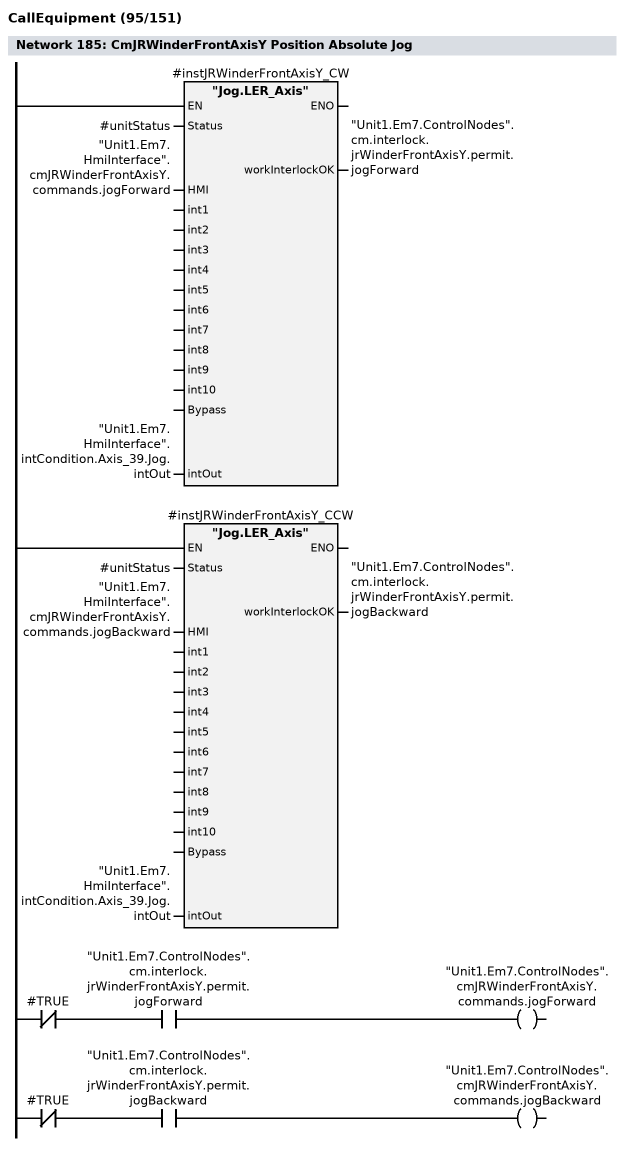
   RUNG wire#powerrail
      #instJRWinderFrontAxisY_CW(Status := #unitStatus, HMI := "Unit1.Em7.HmiInterface".cmJRWinderFrontAxisY.commands.jogForward, int1 :=, int2 :=, int3 :=, int4 :=, int5 :=, int6 :=, int7 :=, int8 :=, int9 :=, int10 :=, Bypass :=, intOut := "Unit1.Em7.HmiInterface".intCondition.Axis_39.Jog.intOut, workInterlockOK => "Unit1.Em7.ControlNodes".cm.interlock.jrWinderFrontAxisY.permit.jogForward)
   END_RUNG
   RUNG wire#powerrail
      #instJRWinderFrontAxisY_CCW(Status := #unitStatus, HMI := "Unit1.Em7.HmiInterface".cmJRWinderFrontAxisY.commands.jogBackward, int1 :=, int2 :=, int3 :=, int4 :=, int5 :=, int6 :=, int7 :=, int8 :=, int9 :=, int10 :=, Bypass :=, intOut := "Unit1.Em7.HmiInterface".intCondition.Axis_39.Jog.intOut, workInterlockOK => "Unit1.Em7.ControlNodes".cm.interlock.jrWinderFrontAxisY.permit.jogBackward)
   END_RUNG
   RUNG wire#powerrail
      I_Contact( #TRUE )
      Contact( "Unit1.Em7.ControlNodes".cm.interlock.jrWinderFrontAxisY.permit.jogForward )
      Coil( "Unit1.Em7.ControlNodes".cmJRWinderFrontAxisY.commands.jogForward )
   END_RUNG
   RUNG wire#powerrail
      I_Contact( #TRUE )
      Contact( "Unit1.Em7.ControlNodes".cm.interlock.jrWinderFrontAxisY.permit.jogBackward )
      Coil( "Unit1.Em7.ControlNodes".cmJRWinderFrontAxisY.commands.jogBackward )
   END_RUNG
   // the same network as SCL:
   #instJRWinderFrontAxisY_CW(Status := #unitStatus,   // "Jog.LER_Axis"
                           HMI := "Unit1.Em7.HmiInterface".cmJRWinderFrontAxisY.commands.jogForward,
                           intOut := "Unit1.Em7.HmiInterface".intCondition.Axis_39.Jog.intOut,
                           workInterlockOK => "Unit1.Em7.ControlNodes".cm.interlock.jrWinderFrontAxisY.permit.jogForward);
   #instJRWinderFrontAxisY_CCW(Status := #unitStatus,   // "Jog.LER_Axis"
                           HMI := "Unit1.Em7.HmiInterface".cmJRWinderFrontAxisY.commands.jogBackward,
                           intOut := "Unit1.Em7.HmiInterface".intCondition.Axis_39.Jog.intOut,
                           workInterlockOK => "Unit1.Em7.ControlNodes".cm.interlock.jrWinderFrontAxisY.permit.jogBackward);
   "Unit1.Em7.ControlNodes".cmJRWinderFrontAxisY.commands.jogForward := NOT #TRUE AND "Unit1.Em7.ControlNodes".cm.interlock.jrWinderFrontAxisY.permit.jogForward;
   "Unit1.Em7.ControlNodes".cmJRWinderFrontAxisY.commands.jogBackward := NOT #TRUE AND "Unit1.Em7.ControlNodes".cm.interlock.jrWinderFrontAxisY.permit.jogBackward;
END_REGION

REGION Network 186: CmJRWinderFrontAxisY Position Absolute Position0
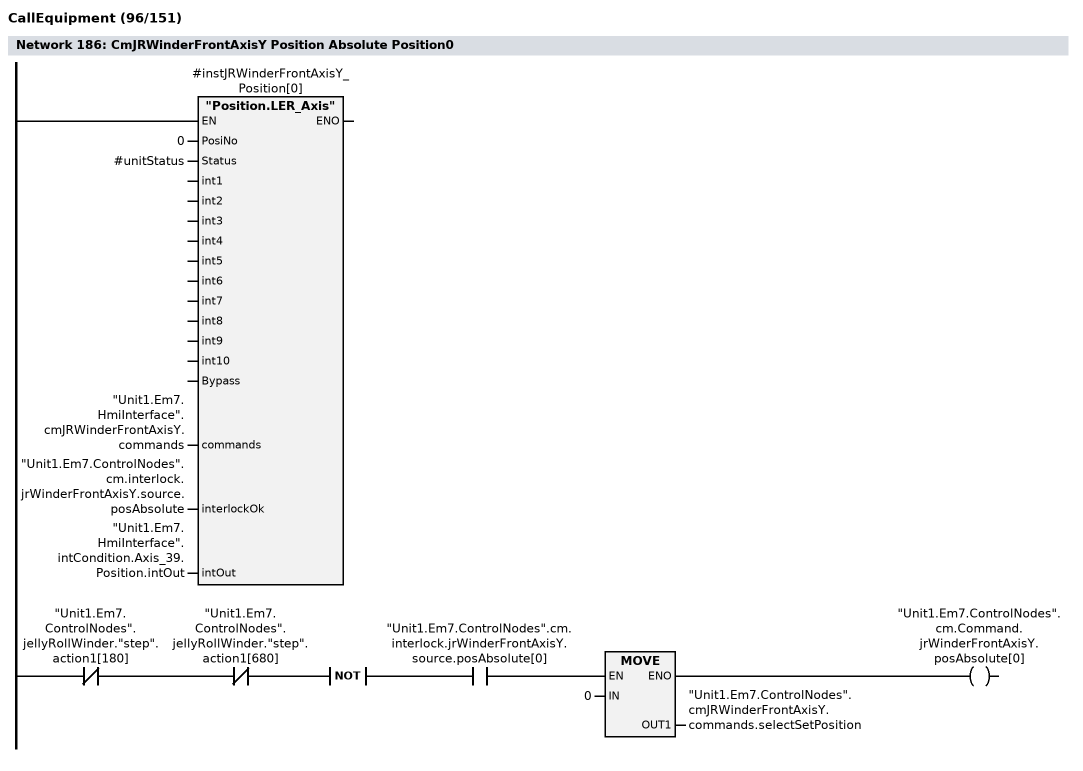
   RUNG wire#powerrail
      #instJRWinderFrontAxisY_Position[0](PosiNo := 0, Status := #unitStatus, int1 :=, int2 :=, int3 :=, int4 :=, int5 :=, int6 :=, int7 :=, int8 :=, int9 :=, int10 :=, Bypass :=, commands := "Unit1.Em7.HmiInterface".cmJRWinderFrontAxisY.commands, interlockOk := "Unit1.Em7.ControlNodes".cm.interlock.jrWinderFrontAxisY.source.posAbsolute, intOut := "Unit1.Em7.HmiInterface".intCondition.Axis_39.Position.intOut)
   END_RUNG
   RUNG wire#powerrail
      I_Contact( "Unit1.Em7.ControlNodes".jellyRollWinder."step".action1[180] )
      I_Contact( "Unit1.Em7.ControlNodes".jellyRollWinder."step".action1[680] )
      Not()
      Contact( "Unit1.Em7.ControlNodes".cm.interlock.jrWinderFrontAxisY.source.posAbsolute[0] )
      Move(in := 0, out1 => "Unit1.Em7.ControlNodes".cmJRWinderFrontAxisY.commands.selectSetPosition)
      Coil( "Unit1.Em7.ControlNodes".cm.Command.jrWinderFrontAxisY.posAbsolute[0] )
   END_RUNG
   // the same network as SCL:
   #instJRWinderFrontAxisY_Position[0](PosiNo := 0,   // "Position.LER_Axis"
                           Status := #unitStatus,
                           commands := "Unit1.Em7.HmiInterface".cmJRWinderFrontAxisY.commands,
                           interlockOk := "Unit1.Em7.ControlNodes".cm.interlock.jrWinderFrontAxisY.source.posAbsolute,
                           intOut := "Unit1.Em7.HmiInterface".intCondition.Axis_39.Position.intOut);
   #_w1 := NOT (NOT "Unit1.Em7.ControlNodes".jellyRollWinder."step".action1[180] AND NOT "Unit1.Em7.ControlNodes".jellyRollWinder."step".action1[680]) AND "Unit1.Em7.ControlNodes".cm.interlock.jrWinderFrontAxisY.source.posAbsolute[0];
   IF #_w1 THEN "Unit1.Em7.ControlNodes".cmJRWinderFrontAxisY.commands.selectSetPosition := 0; END_IF;
   "Unit1.Em7.ControlNodes".cm.Command.jrWinderFrontAxisY.posAbsolute[0] := #_w1;
END_REGION

REGION Network 187: CmJRWinderFrontAxisY Position Absolute Position1
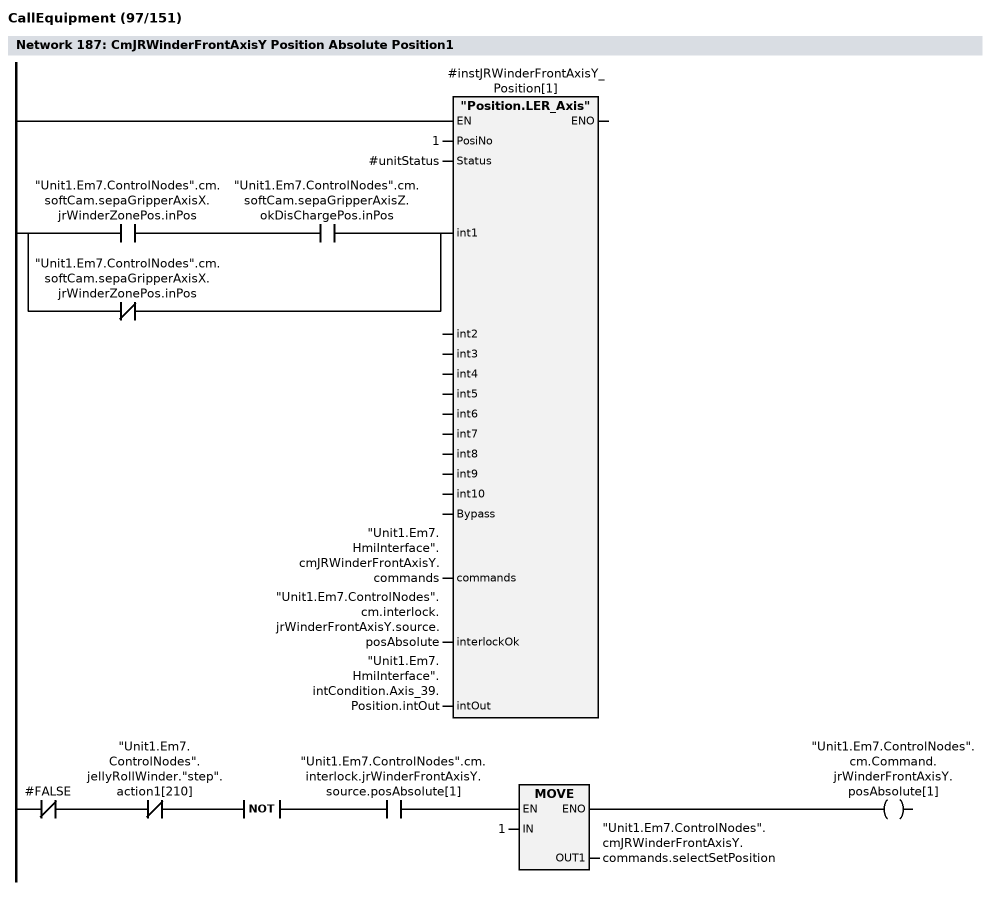
   RUNG wire#powerrail
      #instJRWinderFrontAxisY_Position[1](int1 := wire#w1, PosiNo := 1, Status := #unitStatus, int2 :=, int3 :=, int4 :=, int5 :=, int6 :=, int7 :=, int8 :=, int9 :=, int10 :=, Bypass :=, commands := "Unit1.Em7.HmiInterface".cmJRWinderFrontAxisY.commands, interlockOk := "Unit1.Em7.ControlNodes".cm.interlock.jrWinderFrontAxisY.source.posAbsolute, intOut := "Unit1.Em7.HmiInterface".intCondition.Axis_39.Position.intOut)
   END_RUNG
   RUNG wire#powerrail
      Contact( "Unit1.Em7.ControlNodes".cm.softCam.sepaGripperAxisX.jrWinderZonePos.inPos )
      Contact( "Unit1.Em7.ControlNodes".cm.softCam.sepaGripperAxisZ.okDisChargePos.inPos )
   END_RUNG wire#w1
   RUNG wire#powerrail
      I_Contact( "Unit1.Em7.ControlNodes".cm.softCam.sepaGripperAxisX.jrWinderZonePos.inPos )
   END_RUNG wire#w1
   RUNG wire#powerrail
      I_Contact( #FALSE )
      I_Contact( "Unit1.Em7.ControlNodes".jellyRollWinder."step".action1[210] )
      Not()
      Contact( "Unit1.Em7.ControlNodes".cm.interlock.jrWinderFrontAxisY.source.posAbsolute[1] )
      Move(in := 1, out1 => "Unit1.Em7.ControlNodes".cmJRWinderFrontAxisY.commands.selectSetPosition)
      Coil( "Unit1.Em7.ControlNodes".cm.Command.jrWinderFrontAxisY.posAbsolute[1] )
   END_RUNG
   // the same network as SCL:
   #instJRWinderFrontAxisY_Position[1](PosiNo := 1,   // "Position.LER_Axis"
                           Status := #unitStatus,
                           int1 := ("Unit1.Em7.ControlNodes".cm.softCam.sepaGripperAxisX.jrWinderZonePos.inPos AND "Unit1.Em7.ControlNodes".cm.softCam.sepaGripperAxisZ.okDisChargePos.inPos) OR NOT "Unit1.Em7.ControlNodes".cm.softCam.sepaGripperAxisX.jrWinderZonePos.inPos,
                           commands := "Unit1.Em7.HmiInterface".cmJRWinderFrontAxisY.commands,
                           interlockOk := "Unit1.Em7.ControlNodes".cm.interlock.jrWinderFrontAxisY.source.posAbsolute,
                           intOut := "Unit1.Em7.HmiInterface".intCondition.Axis_39.Position.intOut);
   #_w1 := NOT (NOT #FALSE AND NOT "Unit1.Em7.ControlNodes".jellyRollWinder."step".action1[210]) AND "Unit1.Em7.ControlNodes".cm.interlock.jrWinderFrontAxisY.source.posAbsolute[1];
   IF #_w1 THEN "Unit1.Em7.ControlNodes".cmJRWinderFrontAxisY.commands.selectSetPosition := 1; END_IF;
   "Unit1.Em7.ControlNodes".cm.Command.jrWinderFrontAxisY.posAbsolute[1] := #_w1;
END_REGION

REGION Network 188: CmJRWinderFrontAxisY Position Absolute Position2
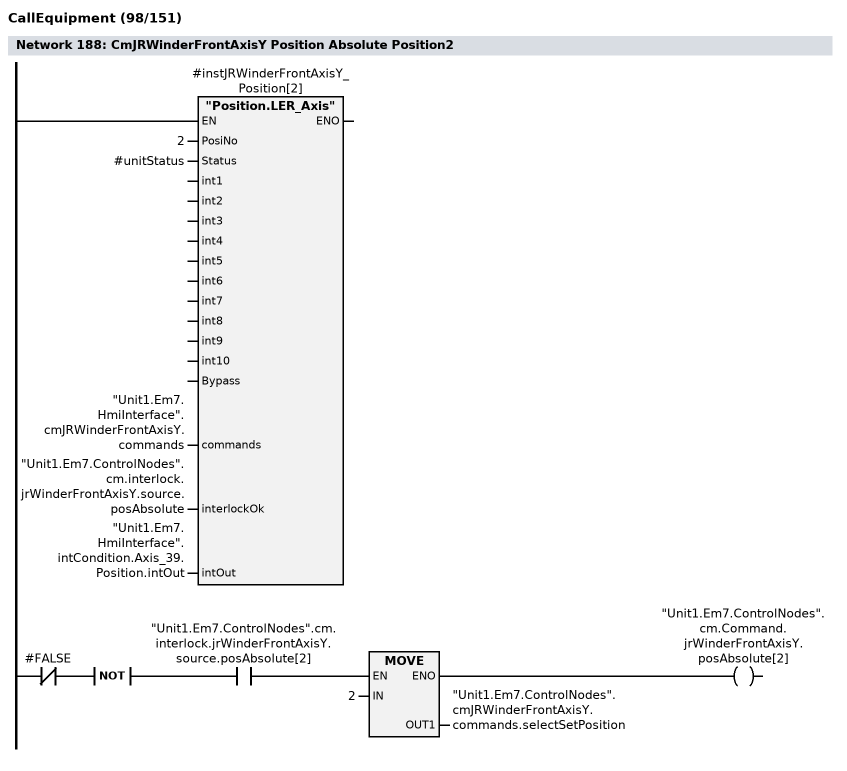
   RUNG wire#powerrail
      #instJRWinderFrontAxisY_Position[2](PosiNo := 2, Status := #unitStatus, int1 :=, int2 :=, int3 :=, int4 :=, int5 :=, int6 :=, int7 :=, int8 :=, int9 :=, int10 :=, Bypass :=, commands := "Unit1.Em7.HmiInterface".cmJRWinderFrontAxisY.commands, interlockOk := "Unit1.Em7.ControlNodes".cm.interlock.jrWinderFrontAxisY.source.posAbsolute, intOut := "Unit1.Em7.HmiInterface".intCondition.Axis_39.Position.intOut)
   END_RUNG
   RUNG wire#powerrail
      I_Contact( #FALSE )
      Not()
      Contact( "Unit1.Em7.ControlNodes".cm.interlock.jrWinderFrontAxisY.source.posAbsolute[2] )
      Move(in := 2, out1 => "Unit1.Em7.ControlNodes".cmJRWinderFrontAxisY.commands.selectSetPosition)
      Coil( "Unit1.Em7.ControlNodes".cm.Command.jrWinderFrontAxisY.posAbsolute[2] )
   END_RUNG
   // the same network as SCL:
   #instJRWinderFrontAxisY_Position[2](PosiNo := 2,   // "Position.LER_Axis"
                           Status := #unitStatus,
                           commands := "Unit1.Em7.HmiInterface".cmJRWinderFrontAxisY.commands,
                           interlockOk := "Unit1.Em7.ControlNodes".cm.interlock.jrWinderFrontAxisY.source.posAbsolute,
                           intOut := "Unit1.Em7.HmiInterface".intCondition.Axis_39.Position.intOut);
   #_w1 := NOT (NOT #FALSE) AND "Unit1.Em7.ControlNodes".cm.interlock.jrWinderFrontAxisY.source.posAbsolute[2];
   IF #_w1 THEN "Unit1.Em7.ControlNodes".cmJRWinderFrontAxisY.commands.selectSetPosition := 2; END_IF;
   "Unit1.Em7.ControlNodes".cm.Command.jrWinderFrontAxisY.posAbsolute[2] := #_w1;
END_REGION

REGION Network 189: CmJRWinderFrontAxisY Position Absolute Position3
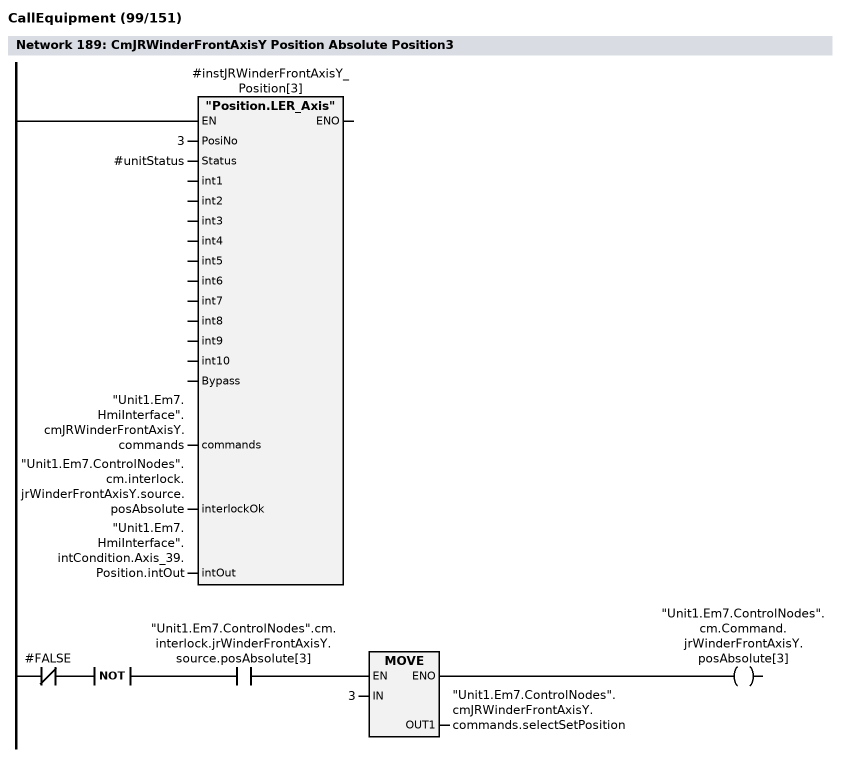
   RUNG wire#powerrail
      #instJRWinderFrontAxisY_Position[3](PosiNo := 3, Status := #unitStatus, int1 :=, int2 :=, int3 :=, int4 :=, int5 :=, int6 :=, int7 :=, int8 :=, int9 :=, int10 :=, Bypass :=, commands := "Unit1.Em7.HmiInterface".cmJRWinderFrontAxisY.commands, interlockOk := "Unit1.Em7.ControlNodes".cm.interlock.jrWinderFrontAxisY.source.posAbsolute, intOut := "Unit1.Em7.HmiInterface".intCondition.Axis_39.Position.intOut)
   END_RUNG
   RUNG wire#powerrail
      I_Contact( #FALSE )
      Not()
      Contact( "Unit1.Em7.ControlNodes".cm.interlock.jrWinderFrontAxisY.source.posAbsolute[3] )
      Move(in := 3, out1 => "Unit1.Em7.ControlNodes".cmJRWinderFrontAxisY.commands.selectSetPosition)
      Coil( "Unit1.Em7.ControlNodes".cm.Command.jrWinderFrontAxisY.posAbsolute[3] )
   END_RUNG
   // the same network as SCL:
   #instJRWinderFrontAxisY_Position[3](PosiNo := 3,   // "Position.LER_Axis"
                           Status := #unitStatus,
                           commands := "Unit1.Em7.HmiInterface".cmJRWinderFrontAxisY.commands,
                           interlockOk := "Unit1.Em7.ControlNodes".cm.interlock.jrWinderFrontAxisY.source.posAbsolute,
                           intOut := "Unit1.Em7.HmiInterface".intCondition.Axis_39.Position.intOut);
   #_w1 := NOT (NOT #FALSE) AND "Unit1.Em7.ControlNodes".cm.interlock.jrWinderFrontAxisY.source.posAbsolute[3];
   IF #_w1 THEN "Unit1.Em7.ControlNodes".cmJRWinderFrontAxisY.commands.selectSetPosition := 3; END_IF;
   "Unit1.Em7.ControlNodes".cm.Command.jrWinderFrontAxisY.posAbsolute[3] := #_w1;
END_REGION

REGION Network 190: CmJRWinderFrontAxisY Position Absolute Position4
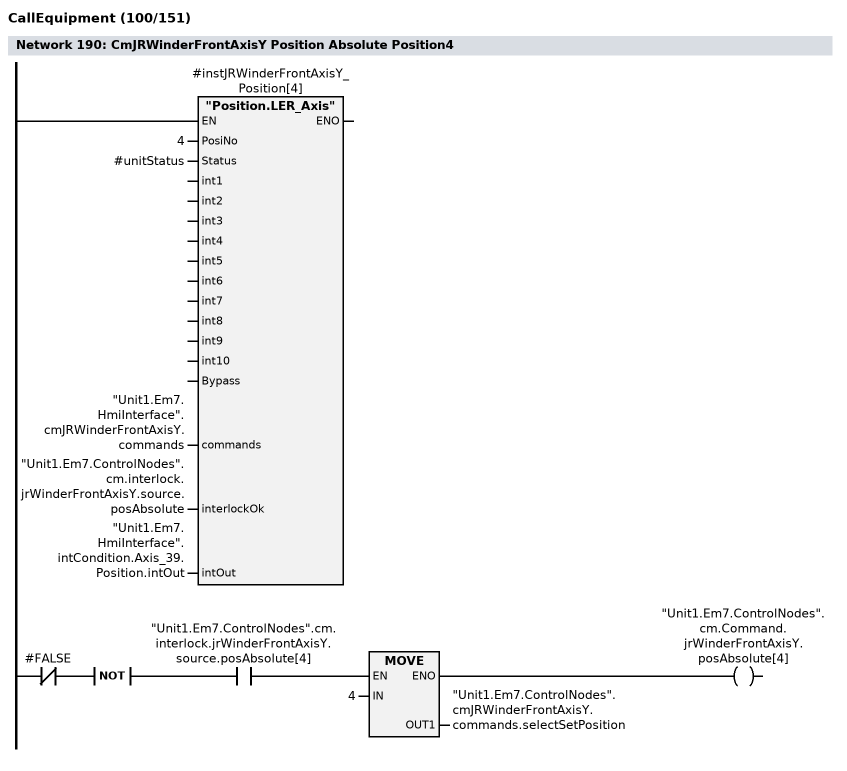
   RUNG wire#powerrail
      #instJRWinderFrontAxisY_Position[4](PosiNo := 4, Status := #unitStatus, int1 :=, int2 :=, int3 :=, int4 :=, int5 :=, int6 :=, int7 :=, int8 :=, int9 :=, int10 :=, Bypass :=, commands := "Unit1.Em7.HmiInterface".cmJRWinderFrontAxisY.commands, interlockOk := "Unit1.Em7.ControlNodes".cm.interlock.jrWinderFrontAxisY.source.posAbsolute, intOut := "Unit1.Em7.HmiInterface".intCondition.Axis_39.Position.intOut)
   END_RUNG
   RUNG wire#powerrail
      I_Contact( #FALSE )
      Not()
      Contact( "Unit1.Em7.ControlNodes".cm.interlock.jrWinderFrontAxisY.source.posAbsolute[4] )
      Move(in := 4, out1 => "Unit1.Em7.ControlNodes".cmJRWinderFrontAxisY.commands.selectSetPosition)
      Coil( "Unit1.Em7.ControlNodes".cm.Command.jrWinderFrontAxisY.posAbsolute[4] )
   END_RUNG
   // the same network as SCL:
   #instJRWinderFrontAxisY_Position[4](PosiNo := 4,   // "Position.LER_Axis"
                           Status := #unitStatus,
                           commands := "Unit1.Em7.HmiInterface".cmJRWinderFrontAxisY.commands,
                           interlockOk := "Unit1.Em7.ControlNodes".cm.interlock.jrWinderFrontAxisY.source.posAbsolute,
                           intOut := "Unit1.Em7.HmiInterface".intCondition.Axis_39.Position.intOut);
   #_w1 := NOT (NOT #FALSE) AND "Unit1.Em7.ControlNodes".cm.interlock.jrWinderFrontAxisY.source.posAbsolute[4];
   IF #_w1 THEN "Unit1.Em7.ControlNodes".cmJRWinderFrontAxisY.commands.selectSetPosition := 4; END_IF;
   "Unit1.Em7.ControlNodes".cm.Command.jrWinderFrontAxisY.posAbsolute[4] := #_w1;
END_REGION

REGION Network 191: CmJRWinderFrontAxisY Position Absolute Position5
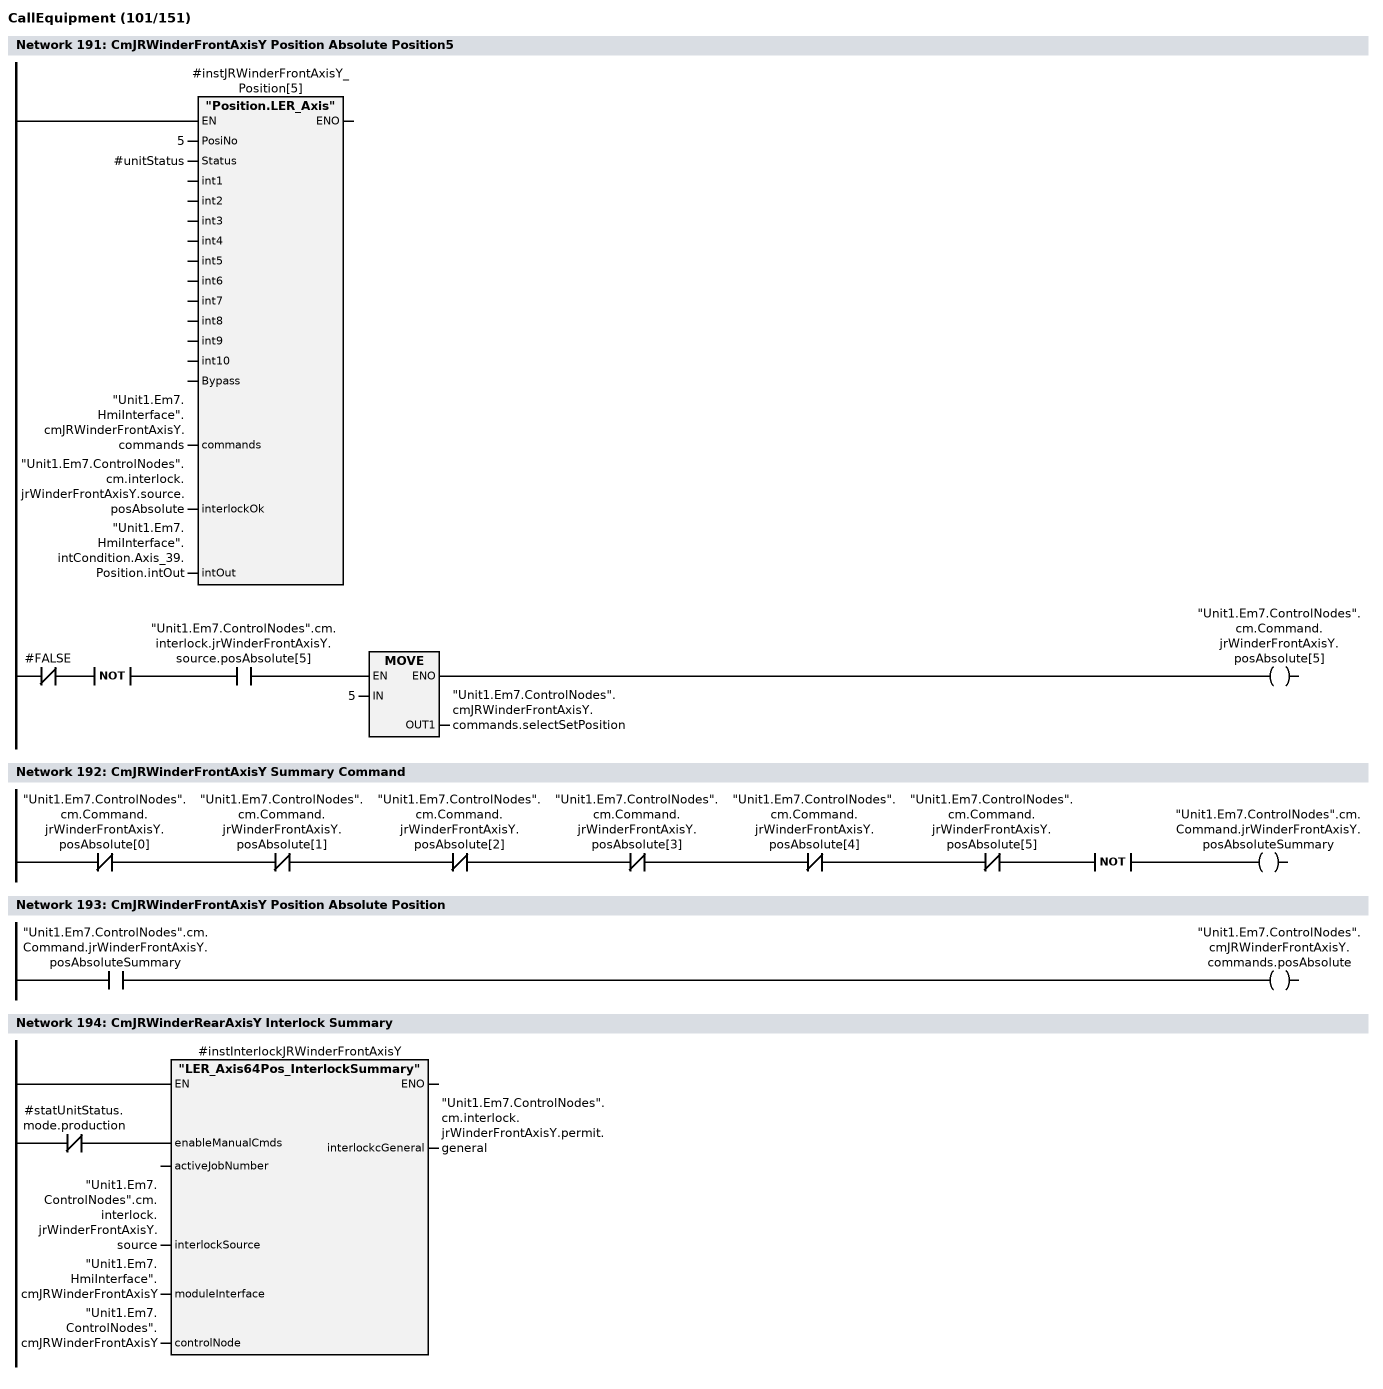
   RUNG wire#powerrail
      #instJRWinderFrontAxisY_Position[5](PosiNo := 5, Status := #unitStatus, int1 :=, int2 :=, int3 :=, int4 :=, int5 :=, int6 :=, int7 :=, int8 :=, int9 :=, int10 :=, Bypass :=, commands := "Unit1.Em7.HmiInterface".cmJRWinderFrontAxisY.commands, interlockOk := "Unit1.Em7.ControlNodes".cm.interlock.jrWinderFrontAxisY.source.posAbsolute, intOut := "Unit1.Em7.HmiInterface".intCondition.Axis_39.Position.intOut)
   END_RUNG
   RUNG wire#powerrail
      I_Contact( #FALSE )
      Not()
      Contact( "Unit1.Em7.ControlNodes".cm.interlock.jrWinderFrontAxisY.source.posAbsolute[5] )
      Move(in := 5, out1 => "Unit1.Em7.ControlNodes".cmJRWinderFrontAxisY.commands.selectSetPosition)
      Coil( "Unit1.Em7.ControlNodes".cm.Command.jrWinderFrontAxisY.posAbsolute[5] )
   END_RUNG
   // the same network as SCL:
   #instJRWinderFrontAxisY_Position[5](PosiNo := 5,   // "Position.LER_Axis"
                           Status := #unitStatus,
                           commands := "Unit1.Em7.HmiInterface".cmJRWinderFrontAxisY.commands,
                           interlockOk := "Unit1.Em7.ControlNodes".cm.interlock.jrWinderFrontAxisY.source.posAbsolute,
                           intOut := "Unit1.Em7.HmiInterface".intCondition.Axis_39.Position.intOut);
   #_w1 := NOT (NOT #FALSE) AND "Unit1.Em7.ControlNodes".cm.interlock.jrWinderFrontAxisY.source.posAbsolute[5];
   IF #_w1 THEN "Unit1.Em7.ControlNodes".cmJRWinderFrontAxisY.commands.selectSetPosition := 5; END_IF;
   "Unit1.Em7.ControlNodes".cm.Command.jrWinderFrontAxisY.posAbsolute[5] := #_w1;
END_REGION

REGION Network 192: CmJRWinderFrontAxisY Summary Command
   RUNG wire#powerrail
      I_Contact( "Unit1.Em7.ControlNodes".cm.Command.jrWinderFrontAxisY.posAbsolute[0] )
      I_Contact( "Unit1.Em7.ControlNodes".cm.Command.jrWinderFrontAxisY.posAbsolute[1] )
      I_Contact( "Unit1.Em7.ControlNodes".cm.Command.jrWinderFrontAxisY.posAbsolute[2] )
      I_Contact( "Unit1.Em7.ControlNodes".cm.Command.jrWinderFrontAxisY.posAbsolute[3] )
      I_Contact( "Unit1.Em7.ControlNodes".cm.Command.jrWinderFrontAxisY.posAbsolute[4] )
      I_Contact( "Unit1.Em7.ControlNodes".cm.Command.jrWinderFrontAxisY.posAbsolute[5] )
      Not()
      Coil( "Unit1.Em7.ControlNodes".cm.Command.jrWinderFrontAxisY.posAbsoluteSummary )
   END_RUNG
   // the same network as SCL:
   "Unit1.Em7.ControlNodes".cm.Command.jrWinderFrontAxisY.posAbsoluteSummary := NOT (NOT "Unit1.Em7.ControlNodes".cm.Command.jrWinderFrontAxisY.posAbsolute[0] AND NOT "Unit1.Em7.ControlNodes".cm.Command.jrWinderFrontAxisY.posAbsolute[1] AND NOT "Unit1.Em7.ControlNodes".cm.Command.jrWinderFrontAxisY.posAbsolute[2] AND NOT "Unit1.Em7.ControlNodes".cm.Command.jrWinderFrontAxisY.posAbsolute[3] AND NOT "Unit1.Em7.ControlNodes".cm.Command.jrWinderFrontAxisY.posAbsolute[4] AND NOT "Unit1.Em7.ControlNodes".cm.Command.jrWinderFrontAxisY.posAbsolute[5]);
END_REGION

REGION Network 193: CmJRWinderFrontAxisY Position Absolute Position
   RUNG wire#powerrail
      Contact( "Unit1.Em7.ControlNodes".cm.Command.jrWinderFrontAxisY.posAbsoluteSummary )
      Coil( "Unit1.Em7.ControlNodes".cmJRWinderFrontAxisY.commands.posAbsolute )
   END_RUNG
   // the same network as SCL:
   "Unit1.Em7.ControlNodes".cmJRWinderFrontAxisY.commands.posAbsolute := "Unit1.Em7.ControlNodes".cm.Command.jrWinderFrontAxisY.posAbsoluteSummary;
END_REGION

REGION Network 194: CmJRWinderRearAxisY Interlock Summary
   RUNG wire#powerrail
      #instInterlockJRWinderFrontAxisY(enableManualCmds := wire#w1, activeJobNumber :=, interlockSource := "Unit1.Em7.ControlNodes".cm.interlock.jrWinderFrontAxisY.source, moduleInterface := "Unit1.Em7.HmiInterface".cmJRWinderFrontAxisY, controlNode := "Unit1.Em7.ControlNodes".cmJRWinderFrontAxisY, interlockcGeneral => "Unit1.Em7.ControlNodes".cm.interlock.jrWinderFrontAxisY.permit.general)
   END_RUNG
   RUNG wire#powerrail
      I_Contact( #statUnitStatus.mode.production )
   END_RUNG wire#w1
   // the same network as SCL:
   #instInterlockJRWinderFrontAxisY(enableManualCmds := NOT #statUnitStatus.mode.production,   // "LER_Axis64Pos_InterlockSummary"
                           interlockSource := "Unit1.Em7.ControlNodes".cm.interlock.jrWinderFrontAxisY.source,
                           moduleInterface := "Unit1.Em7.HmiInterface".cmJRWinderFrontAxisY,
                           controlNode := "Unit1.Em7.ControlNodes".cmJRWinderFrontAxisY,
                           interlockcGeneral => "Unit1.Em7.ControlNodes".cm.interlock.jrWinderFrontAxisY.permit.general);
END_REGION

REGION Network 195: CmJRWinderFrontAxisY velocity/speed
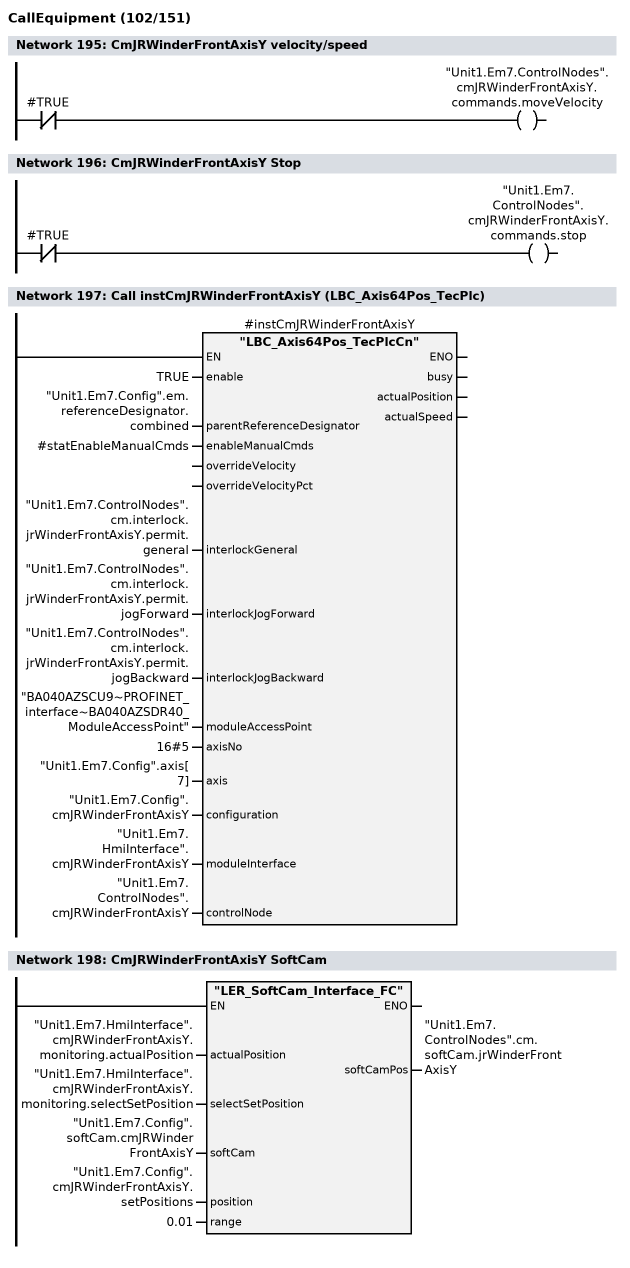
   RUNG wire#powerrail
      I_Contact( #TRUE )
      Coil( "Unit1.Em7.ControlNodes".cmJRWinderFrontAxisY.commands.moveVelocity )
   END_RUNG
   // the same network as SCL:
   "Unit1.Em7.ControlNodes".cmJRWinderFrontAxisY.commands.moveVelocity := NOT #TRUE;
END_REGION

REGION Network 196: CmJRWinderFrontAxisY Stop
   RUNG wire#powerrail
      I_Contact( #TRUE )
      Coil( "Unit1.Em7.ControlNodes".cmJRWinderFrontAxisY.commands.stop )
   END_RUNG
   // the same network as SCL:
   "Unit1.Em7.ControlNodes".cmJRWinderFrontAxisY.commands.stop := NOT #TRUE;
END_REGION

REGION Network 197: Call instCmJRWinderFrontAxisY (LBC_Axis64Pos_TecPlc)
   RUNG wire#powerrail
      #instCmJRWinderFrontAxisY(enable := TRUE, parentReferenceDesignator := "Unit1.Em7.Config".em.referenceDesignator.combined, enableManualCmds := #statEnableManualCmds, overrideVelocity :=, overrideVelocityPct :=, interlockGeneral := "Unit1.Em7.ControlNodes".cm.interlock.jrWinderFrontAxisY.permit.general, interlockJogForward := "Unit1.Em7.ControlNodes".cm.interlock.jrWinderFrontAxisY.permit.jogForward, interlockJogBackward := "Unit1.Em7.ControlNodes".cm.interlock.jrWinderFrontAxisY.permit.jogBackward, moduleAccessPoint := "BA040AZSCU9~PROFINET_interface~BA040AZSDR40_ModuleAccessPoint", axisNo := 16#5, axis := "Unit1.Em7.Config".axis[7], configuration := "Unit1.Em7.Config".cmJRWinderFrontAxisY, moduleInterface := "Unit1.Em7.HmiInterface".cmJRWinderFrontAxisY, controlNode := "Unit1.Em7.ControlNodes".cmJRWinderFrontAxisY, busy =>, actualPosition =>, actualSpeed =>)
   END_RUNG
   // the same network as SCL:
   #instCmJRWinderFrontAxisY(enable := TRUE,   // "LBC_Axis64Pos_TecPlcCn"
                           parentReferenceDesignator := "Unit1.Em7.Config".em.referenceDesignator.combined,
                           enableManualCmds := #statEnableManualCmds,
                           interlockGeneral := "Unit1.Em7.ControlNodes".cm.interlock.jrWinderFrontAxisY.permit.general,
                           interlockJogForward := "Unit1.Em7.ControlNodes".cm.interlock.jrWinderFrontAxisY.permit.jogForward,
                           interlockJogBackward := "Unit1.Em7.ControlNodes".cm.interlock.jrWinderFrontAxisY.permit.jogBackward,
                           moduleAccessPoint := "BA040AZSCU9~PROFINET_interface~BA040AZSDR40_ModuleAccessPoint",
                           axisNo := 16#5,
                           axis := "Unit1.Em7.Config".axis[7],
                           configuration := "Unit1.Em7.Config".cmJRWinderFrontAxisY,
                           moduleInterface := "Unit1.Em7.HmiInterface".cmJRWinderFrontAxisY,
                           controlNode := "Unit1.Em7.ControlNodes".cmJRWinderFrontAxisY);
END_REGION

REGION Network 198: CmJRWinderFrontAxisY SoftCam
   RUNG wire#powerrail
      "LER_SoftCam_Interface_FC"(actualPosition := "Unit1.Em7.HmiInterface".cmJRWinderFrontAxisY.monitoring.actualPosition, selectSetPosition := "Unit1.Em7.HmiInterface".cmJRWinderFrontAxisY.monitoring.selectSetPosition, softCam := "Unit1.Em7.Config".softCam.cmJRWinderFrontAxisY, position := "Unit1.Em7.Config".cmJRWinderFrontAxisY.setPositions, range := 0.01, softCamPos => "Unit1.Em7.ControlNodes".cm.softCam.jrWinderFrontAxisY)
   END_RUNG
   // the same network as SCL:
   "LER_SoftCam_Interface_FC"(actualPosition := "Unit1.Em7.HmiInterface".cmJRWinderFrontAxisY.monitoring.actualPosition,
                           selectSetPosition := "Unit1.Em7.HmiInterface".cmJRWinderFrontAxisY.monitoring.selectSetPosition,
                           softCam := "Unit1.Em7.Config".softCam.cmJRWinderFrontAxisY,
                           position := "Unit1.Em7.Config".cmJRWinderFrontAxisY.setPositions,
                           range := 0.01,
                           softCamPos => "Unit1.Em7.ControlNodes".cm.softCam.jrWinderFrontAxisY);
END_REGION

REGION Network 200: JRWinderAxisB Enable
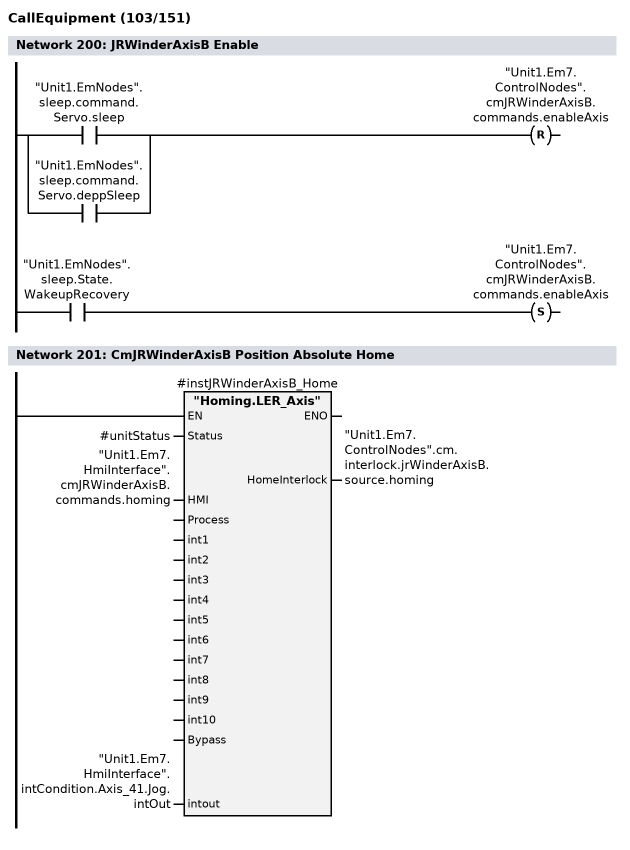
   RUNG wire#powerrail
      Contact( "Unit1.EmNodes".sleep.command.Servo.sleep )
      wire#w1
      R_Coil( "Unit1.Em7.ControlNodes".cmJRWinderAxisB.commands.enableAxis )
   END_RUNG
   RUNG wire#powerrail
      Contact( "Unit1.EmNodes".sleep.command.Servo.deppSleep )
   END_RUNG wire#w1
   RUNG wire#powerrail
      Contact( "Unit1.EmNodes".sleep.State.WakeupRecovery )
      S_Coil( "Unit1.Em7.ControlNodes".cmJRWinderAxisB.commands.enableAxis )
   END_RUNG
   // the same network as SCL:
   IF "Unit1.EmNodes".sleep.command.Servo.sleep OR "Unit1.EmNodes".sleep.command.Servo.deppSleep THEN
       "Unit1.Em7.ControlNodes".cmJRWinderAxisB.commands.enableAxis := FALSE;
   END_IF;
   IF "Unit1.EmNodes".sleep.State.WakeupRecovery THEN
       "Unit1.Em7.ControlNodes".cmJRWinderAxisB.commands.enableAxis := TRUE;
   END_IF;
END_REGION

REGION Network 201: CmJRWinderAxisB Position Absolute Home
   RUNG wire#powerrail
      #instJRWinderAxisB_Home(Status := #unitStatus, HMI := "Unit1.Em7.HmiInterface".cmJRWinderAxisB.commands.homing, Process :=, int1 :=, int2 :=, int3 :=, int4 :=, int5 :=, int6 :=, int7 :=, int8 :=, int9 :=, int10 :=, Bypass :=, intout := "Unit1.Em7.HmiInterface".intCondition.Axis_41.Jog.intOut, HomeInterlock => "Unit1.Em7.ControlNodes".cm.interlock.jrWinderAxisB.source.homing)
   END_RUNG
   // the same network as SCL:
   #instJRWinderAxisB_Home(Status := #unitStatus,   // "Homing.LER_Axis"
                           HMI := "Unit1.Em7.HmiInterface".cmJRWinderAxisB.commands.homing,
                           intout := "Unit1.Em7.HmiInterface".intCondition.Axis_41.Jog.intOut,
                           HomeInterlock => "Unit1.Em7.ControlNodes".cm.interlock.jrWinderAxisB.source.homing);
END_REGION

REGION Network 202: CmJRWinderAxisB Position Absolute Jog
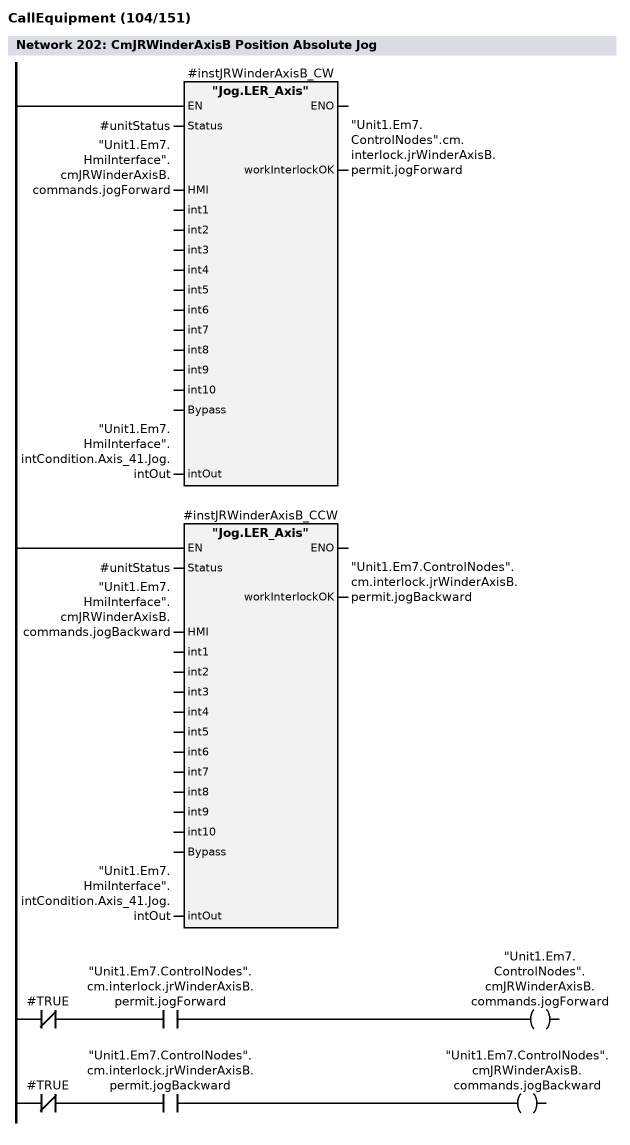
   RUNG wire#powerrail
      #instJRWinderAxisB_CW(Status := #unitStatus, HMI := "Unit1.Em7.HmiInterface".cmJRWinderAxisB.commands.jogForward, int1 :=, int2 :=, int3 :=, int4 :=, int5 :=, int6 :=, int7 :=, int8 :=, int9 :=, int10 :=, Bypass :=, intOut := "Unit1.Em7.HmiInterface".intCondition.Axis_41.Jog.intOut, workInterlockOK => "Unit1.Em7.ControlNodes".cm.interlock.jrWinderAxisB.permit.jogForward)
   END_RUNG
   RUNG wire#powerrail
      #instJRWinderAxisB_CCW(Status := #unitStatus, HMI := "Unit1.Em7.HmiInterface".cmJRWinderAxisB.commands.jogBackward, int1 :=, int2 :=, int3 :=, int4 :=, int5 :=, int6 :=, int7 :=, int8 :=, int9 :=, int10 :=, Bypass :=, intOut := "Unit1.Em7.HmiInterface".intCondition.Axis_41.Jog.intOut, workInterlockOK => "Unit1.Em7.ControlNodes".cm.interlock.jrWinderAxisB.permit.jogBackward)
   END_RUNG
   RUNG wire#powerrail
      I_Contact( #TRUE )
      Contact( "Unit1.Em7.ControlNodes".cm.interlock.jrWinderAxisB.permit.jogForward )
      Coil( "Unit1.Em7.ControlNodes".cmJRWinderAxisB.commands.jogForward )
   END_RUNG
   RUNG wire#powerrail
      I_Contact( #TRUE )
      Contact( "Unit1.Em7.ControlNodes".cm.interlock.jrWinderAxisB.permit.jogBackward )
      Coil( "Unit1.Em7.ControlNodes".cmJRWinderAxisB.commands.jogBackward )
   END_RUNG
   // the same network as SCL:
   #instJRWinderAxisB_CW(Status := #unitStatus,   // "Jog.LER_Axis"
                         HMI := "Unit1.Em7.HmiInterface".cmJRWinderAxisB.commands.jogForward,
                         intOut := "Unit1.Em7.HmiInterface".intCondition.Axis_41.Jog.intOut,
                         workInterlockOK => "Unit1.Em7.ControlNodes".cm.interlock.jrWinderAxisB.permit.jogForward);
   #instJRWinderAxisB_CCW(Status := #unitStatus,   // "Jog.LER_Axis"
                          HMI := "Unit1.Em7.HmiInterface".cmJRWinderAxisB.commands.jogBackward,
                          intOut := "Unit1.Em7.HmiInterface".intCondition.Axis_41.Jog.intOut,
                          workInterlockOK => "Unit1.Em7.ControlNodes".cm.interlock.jrWinderAxisB.permit.jogBackward);
   "Unit1.Em7.ControlNodes".cmJRWinderAxisB.commands.jogForward := NOT #TRUE AND "Unit1.Em7.ControlNodes".cm.interlock.jrWinderAxisB.permit.jogForward;
   "Unit1.Em7.ControlNodes".cmJRWinderAxisB.commands.jogBackward := NOT #TRUE AND "Unit1.Em7.ControlNodes".cm.interlock.jrWinderAxisB.permit.jogBackward;
END_REGION

REGION Network 203: CmJRWinderAxisB Position Absolute Position0
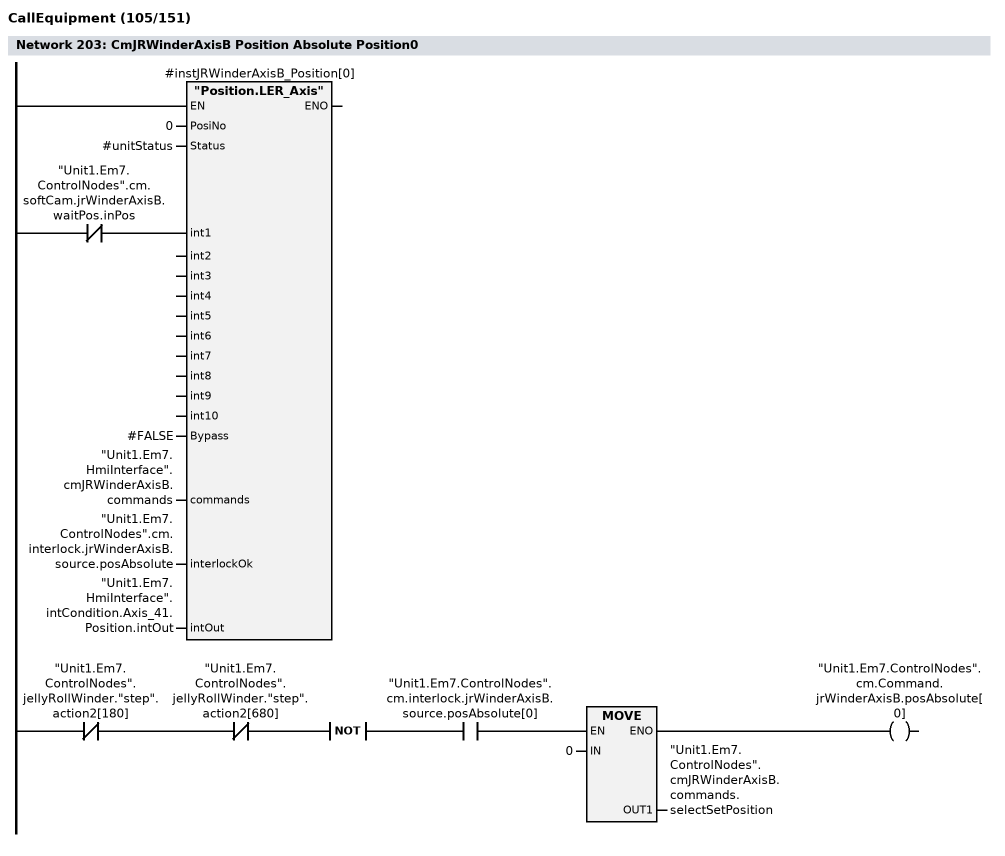
   RUNG wire#powerrail
      #instJRWinderAxisB_Position[0](int1 := wire#w1, PosiNo := 0, Status := #unitStatus, int2 :=, int3 :=, int4 :=, int5 :=, int6 :=, int7 :=, int8 :=, int9 :=, int10 :=, Bypass := #FALSE, commands := "Unit1.Em7.HmiInterface".cmJRWinderAxisB.commands, interlockOk := "Unit1.Em7.ControlNodes".cm.interlock.jrWinderAxisB.source.posAbsolute, intOut := "Unit1.Em7.HmiInterface".intCondition.Axis_41.Position.intOut)
   END_RUNG
   RUNG wire#powerrail
      I_Contact( "Unit1.Em7.ControlNodes".cm.softCam.jrWinderAxisB.waitPos.inPos )
   END_RUNG wire#w1
   RUNG wire#powerrail
      I_Contact( "Unit1.Em7.ControlNodes".jellyRollWinder."step".action2[180] )
      I_Contact( "Unit1.Em7.ControlNodes".jellyRollWinder."step".action2[680] )
      Not()
      Contact( "Unit1.Em7.ControlNodes".cm.interlock.jrWinderAxisB.source.posAbsolute[0] )
      Move(in := 0, out1 => "Unit1.Em7.ControlNodes".cmJRWinderAxisB.commands.selectSetPosition)
      Coil( "Unit1.Em7.ControlNodes".cm.Command.jrWinderAxisB.posAbsolute[0] )
   END_RUNG
   // the same network as SCL:
   #instJRWinderAxisB_Position[0](PosiNo := 0,   // "Position.LER_Axis"
                           Status := #unitStatus,
                           int1 := NOT "Unit1.Em7.ControlNodes".cm.softCam.jrWinderAxisB.waitPos.inPos,
                           Bypass := #FALSE,
                           commands := "Unit1.Em7.HmiInterface".cmJRWinderAxisB.commands,
                           interlockOk := "Unit1.Em7.ControlNodes".cm.interlock.jrWinderAxisB.source.posAbsolute,
                           intOut := "Unit1.Em7.HmiInterface".intCondition.Axis_41.Position.intOut);
   #_w1 := NOT (NOT "Unit1.Em7.ControlNodes".jellyRollWinder."step".action2[180] AND NOT "Unit1.Em7.ControlNodes".jellyRollWinder."step".action2[680]) AND "Unit1.Em7.ControlNodes".cm.interlock.jrWinderAxisB.source.posAbsolute[0];
   IF #_w1 THEN "Unit1.Em7.ControlNodes".cmJRWinderAxisB.commands.selectSetPosition := 0; END_IF;
   "Unit1.Em7.ControlNodes".cm.Command.jrWinderAxisB.posAbsolute[0] := #_w1;
END_REGION

REGION Network 204: CmJRWinderAxisB Position Absolute Position1
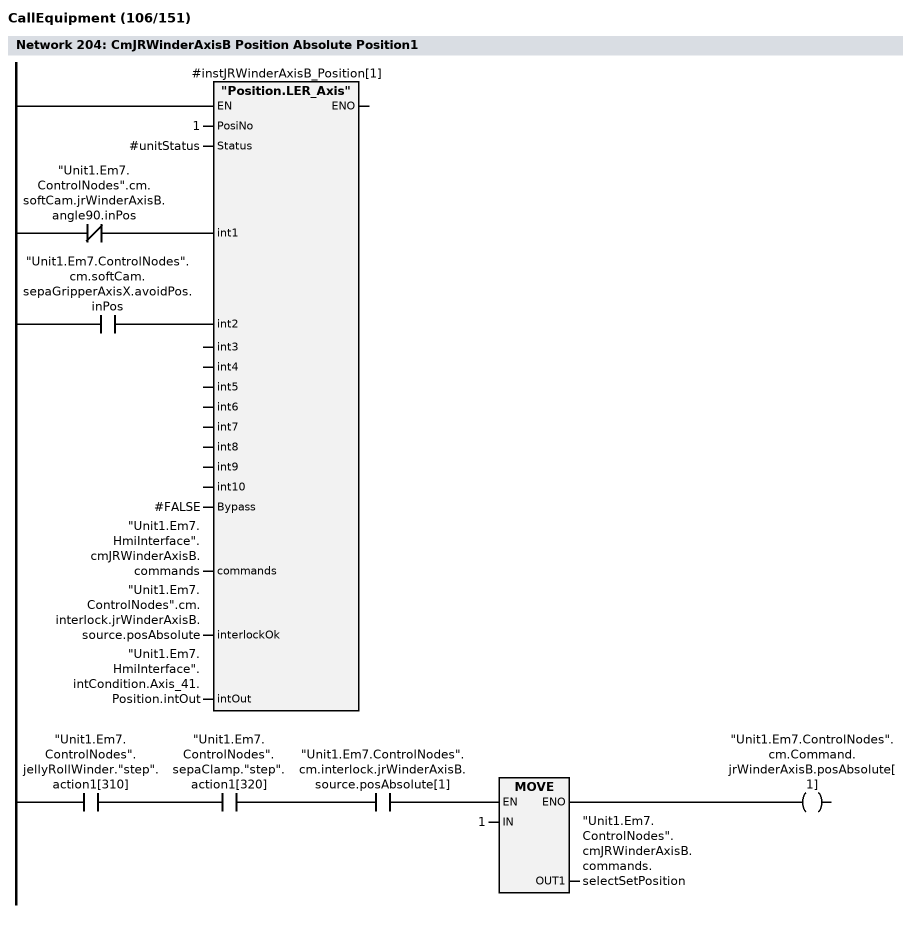
   RUNG wire#powerrail
      #instJRWinderAxisB_Position[1](int1 := wire#w1, int2 := wire#w2, PosiNo := 1, Status := #unitStatus, int3 :=, int4 :=, int5 :=, int6 :=, int7 :=, int8 :=, int9 :=, int10 :=, Bypass := #FALSE, commands := "Unit1.Em7.HmiInterface".cmJRWinderAxisB.commands, interlockOk := "Unit1.Em7.ControlNodes".cm.interlock.jrWinderAxisB.source.posAbsolute, intOut := "Unit1.Em7.HmiInterface".intCondition.Axis_41.Position.intOut)
   END_RUNG
   RUNG wire#powerrail
      I_Contact( "Unit1.Em7.ControlNodes".cm.softCam.jrWinderAxisB.angle90.inPos )
   END_RUNG wire#w1
   RUNG wire#powerrail
      Contact( "Unit1.Em7.ControlNodes".cm.softCam.sepaGripperAxisX.avoidPos.inPos )
   END_RUNG wire#w2
   RUNG wire#powerrail
      Contact( "Unit1.Em7.ControlNodes".jellyRollWinder."step".action1[310] )
      Contact( "Unit1.Em7.ControlNodes".sepaClamp."step".action1[320] )
      Contact( "Unit1.Em7.ControlNodes".cm.interlock.jrWinderAxisB.source.posAbsolute[1] )
      Move(in := 1, out1 => "Unit1.Em7.ControlNodes".cmJRWinderAxisB.commands.selectSetPosition)
      Coil( "Unit1.Em7.ControlNodes".cm.Command.jrWinderAxisB.posAbsolute[1] )
   END_RUNG
   // the same network as SCL:
   #instJRWinderAxisB_Position[1](PosiNo := 1,   // "Position.LER_Axis"
                           Status := #unitStatus,
                           int1 := NOT "Unit1.Em7.ControlNodes".cm.softCam.jrWinderAxisB.angle90.inPos,
                           int2 := "Unit1.Em7.ControlNodes".cm.softCam.sepaGripperAxisX.avoidPos.inPos,
                           Bypass := #FALSE,
                           commands := "Unit1.Em7.HmiInterface".cmJRWinderAxisB.commands,
                           interlockOk := "Unit1.Em7.ControlNodes".cm.interlock.jrWinderAxisB.source.posAbsolute,
                           intOut := "Unit1.Em7.HmiInterface".intCondition.Axis_41.Position.intOut);
   #_w1 := "Unit1.Em7.ControlNodes".jellyRollWinder."step".action1[310] AND "Unit1.Em7.ControlNodes".sepaClamp."step".action1[320] AND "Unit1.Em7.ControlNodes".cm.interlock.jrWinderAxisB.source.posAbsolute[1];
   IF #_w1 THEN "Unit1.Em7.ControlNodes".cmJRWinderAxisB.commands.selectSetPosition := 1; END_IF;
   "Unit1.Em7.ControlNodes".cm.Command.jrWinderAxisB.posAbsolute[1] := #_w1;
END_REGION

REGION Network 205: CmJRWinderAxisB Position Absolute Position2
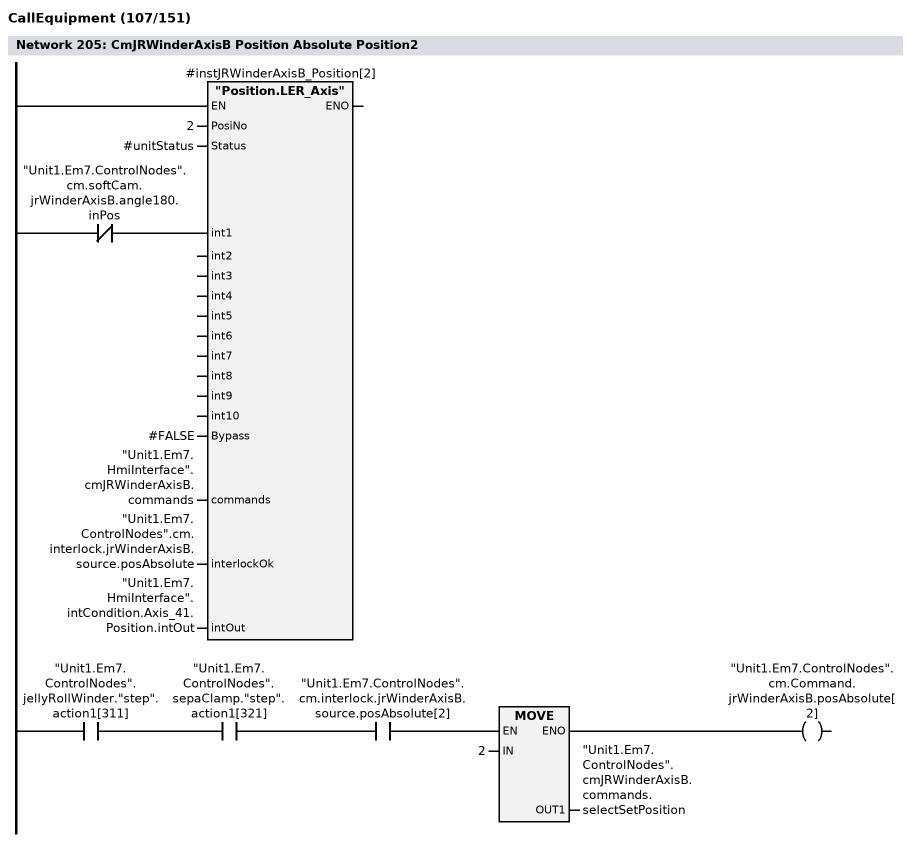
   RUNG wire#powerrail
      #instJRWinderAxisB_Position[2](int1 := wire#w1, PosiNo := 2, Status := #unitStatus, int2 :=, int3 :=, int4 :=, int5 :=, int6 :=, int7 :=, int8 :=, int9 :=, int10 :=, Bypass := #FALSE, commands := "Unit1.Em7.HmiInterface".cmJRWinderAxisB.commands, interlockOk := "Unit1.Em7.ControlNodes".cm.interlock.jrWinderAxisB.source.posAbsolute, intOut := "Unit1.Em7.HmiInterface".intCondition.Axis_41.Position.intOut)
   END_RUNG
   RUNG wire#powerrail
      I_Contact( "Unit1.Em7.ControlNodes".cm.softCam.jrWinderAxisB.angle180.inPos )
   END_RUNG wire#w1
   RUNG wire#powerrail
      Contact( "Unit1.Em7.ControlNodes".jellyRollWinder."step".action1[311] )
      Contact( "Unit1.Em7.ControlNodes".sepaClamp."step".action1[321] )
      Contact( "Unit1.Em7.ControlNodes".cm.interlock.jrWinderAxisB.source.posAbsolute[2] )
      Move(in := 2, out1 => "Unit1.Em7.ControlNodes".cmJRWinderAxisB.commands.selectSetPosition)
      Coil( "Unit1.Em7.ControlNodes".cm.Command.jrWinderAxisB.posAbsolute[2] )
   END_RUNG
   // the same network as SCL:
   #instJRWinderAxisB_Position[2](PosiNo := 2,   // "Position.LER_Axis"
                           Status := #unitStatus,
                           int1 := NOT "Unit1.Em7.ControlNodes".cm.softCam.jrWinderAxisB.angle180.inPos,
                           Bypass := #FALSE,
                           commands := "Unit1.Em7.HmiInterface".cmJRWinderAxisB.commands,
                           interlockOk := "Unit1.Em7.ControlNodes".cm.interlock.jrWinderAxisB.source.posAbsolute,
                           intOut := "Unit1.Em7.HmiInterface".intCondition.Axis_41.Position.intOut);
   #_w1 := "Unit1.Em7.ControlNodes".jellyRollWinder."step".action1[311] AND "Unit1.Em7.ControlNodes".sepaClamp."step".action1[321] AND "Unit1.Em7.ControlNodes".cm.interlock.jrWinderAxisB.source.posAbsolute[2];
   IF #_w1 THEN "Unit1.Em7.ControlNodes".cmJRWinderAxisB.commands.selectSetPosition := 2; END_IF;
   "Unit1.Em7.ControlNodes".cm.Command.jrWinderAxisB.posAbsolute[2] := #_w1;
END_REGION

REGION Network 206: CmJRWinderAxisB Position Absolute Position3
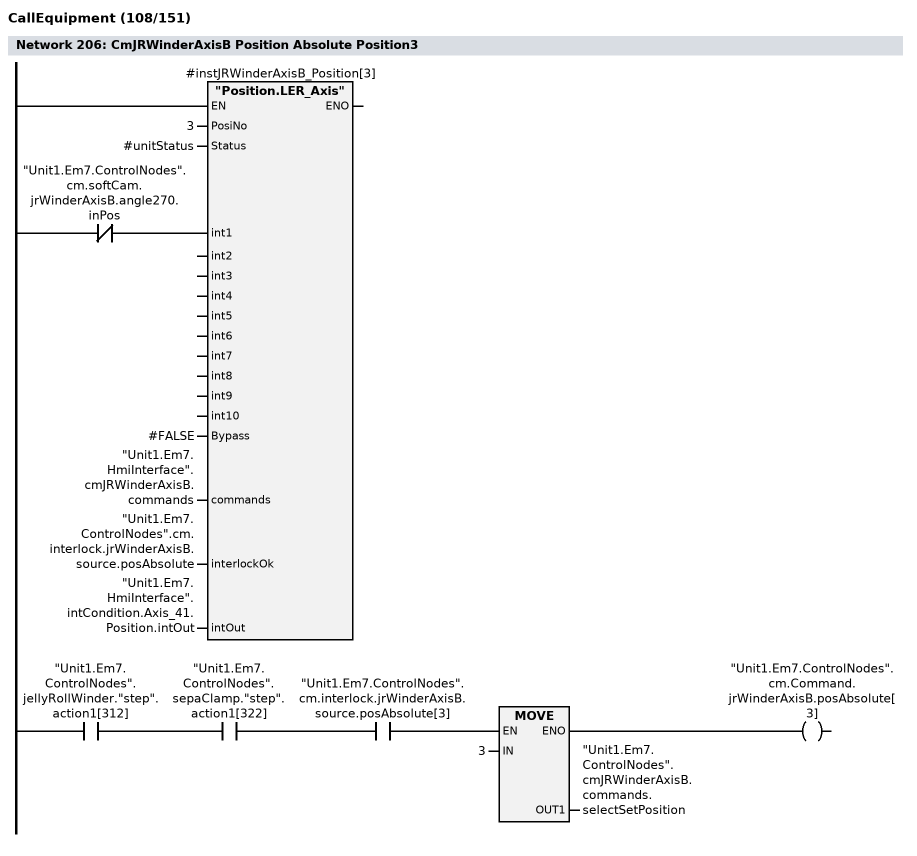
   RUNG wire#powerrail
      #instJRWinderAxisB_Position[3](int1 := wire#w1, PosiNo := 3, Status := #unitStatus, int2 :=, int3 :=, int4 :=, int5 :=, int6 :=, int7 :=, int8 :=, int9 :=, int10 :=, Bypass := #FALSE, commands := "Unit1.Em7.HmiInterface".cmJRWinderAxisB.commands, interlockOk := "Unit1.Em7.ControlNodes".cm.interlock.jrWinderAxisB.source.posAbsolute, intOut := "Unit1.Em7.HmiInterface".intCondition.Axis_41.Position.intOut)
   END_RUNG
   RUNG wire#powerrail
      I_Contact( "Unit1.Em7.ControlNodes".cm.softCam.jrWinderAxisB.angle270.inPos )
   END_RUNG wire#w1
   RUNG wire#powerrail
      Contact( "Unit1.Em7.ControlNodes".jellyRollWinder."step".action1[312] )
      Contact( "Unit1.Em7.ControlNodes".sepaClamp."step".action1[322] )
      Contact( "Unit1.Em7.ControlNodes".cm.interlock.jrWinderAxisB.source.posAbsolute[3] )
      Move(in := 3, out1 => "Unit1.Em7.ControlNodes".cmJRWinderAxisB.commands.selectSetPosition)
      Coil( "Unit1.Em7.ControlNodes".cm.Command.jrWinderAxisB.posAbsolute[3] )
   END_RUNG
   // the same network as SCL:
   #instJRWinderAxisB_Position[3](PosiNo := 3,   // "Position.LER_Axis"
                           Status := #unitStatus,
                           int1 := NOT "Unit1.Em7.ControlNodes".cm.softCam.jrWinderAxisB.angle270.inPos,
                           Bypass := #FALSE,
                           commands := "Unit1.Em7.HmiInterface".cmJRWinderAxisB.commands,
                           interlockOk := "Unit1.Em7.ControlNodes".cm.interlock.jrWinderAxisB.source.posAbsolute,
                           intOut := "Unit1.Em7.HmiInterface".intCondition.Axis_41.Position.intOut);
   #_w1 := "Unit1.Em7.ControlNodes".jellyRollWinder."step".action1[312] AND "Unit1.Em7.ControlNodes".sepaClamp."step".action1[322] AND "Unit1.Em7.ControlNodes".cm.interlock.jrWinderAxisB.source.posAbsolute[3];
   IF #_w1 THEN "Unit1.Em7.ControlNodes".cmJRWinderAxisB.commands.selectSetPosition := 3; END_IF;
   "Unit1.Em7.ControlNodes".cm.Command.jrWinderAxisB.posAbsolute[3] := #_w1;
END_REGION

REGION Network 207: CmJRWinderAxisB Position Absolute Position4
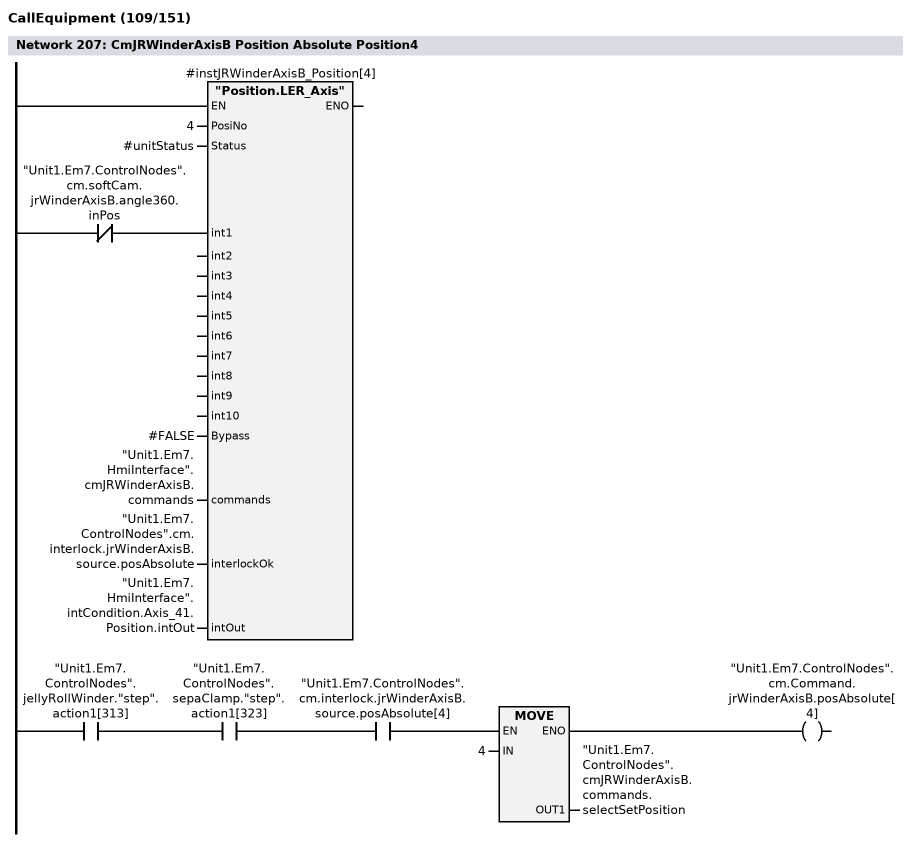
   RUNG wire#powerrail
      #instJRWinderAxisB_Position[4](int1 := wire#w1, PosiNo := 4, Status := #unitStatus, int2 :=, int3 :=, int4 :=, int5 :=, int6 :=, int7 :=, int8 :=, int9 :=, int10 :=, Bypass := #FALSE, commands := "Unit1.Em7.HmiInterface".cmJRWinderAxisB.commands, interlockOk := "Unit1.Em7.ControlNodes".cm.interlock.jrWinderAxisB.source.posAbsolute, intOut := "Unit1.Em7.HmiInterface".intCondition.Axis_41.Position.intOut)
   END_RUNG
   RUNG wire#powerrail
      I_Contact( "Unit1.Em7.ControlNodes".cm.softCam.jrWinderAxisB.angle360.inPos )
   END_RUNG wire#w1
   RUNG wire#powerrail
      Contact( "Unit1.Em7.ControlNodes".jellyRollWinder."step".action1[313] )
      Contact( "Unit1.Em7.ControlNodes".sepaClamp."step".action1[323] )
      Contact( "Unit1.Em7.ControlNodes".cm.interlock.jrWinderAxisB.source.posAbsolute[4] )
      Move(in := 4, out1 => "Unit1.Em7.ControlNodes".cmJRWinderAxisB.commands.selectSetPosition)
      Coil( "Unit1.Em7.ControlNodes".cm.Command.jrWinderAxisB.posAbsolute[4] )
   END_RUNG
   // the same network as SCL:
   #instJRWinderAxisB_Position[4](PosiNo := 4,   // "Position.LER_Axis"
                           Status := #unitStatus,
                           int1 := NOT "Unit1.Em7.ControlNodes".cm.softCam.jrWinderAxisB.angle360.inPos,
                           Bypass := #FALSE,
                           commands := "Unit1.Em7.HmiInterface".cmJRWinderAxisB.commands,
                           interlockOk := "Unit1.Em7.ControlNodes".cm.interlock.jrWinderAxisB.source.posAbsolute,
                           intOut := "Unit1.Em7.HmiInterface".intCondition.Axis_41.Position.intOut);
   #_w1 := "Unit1.Em7.ControlNodes".jellyRollWinder."step".action1[313] AND "Unit1.Em7.ControlNodes".sepaClamp."step".action1[323] AND "Unit1.Em7.ControlNodes".cm.interlock.jrWinderAxisB.source.posAbsolute[4];
   IF #_w1 THEN "Unit1.Em7.ControlNodes".cmJRWinderAxisB.commands.selectSetPosition := 4; END_IF;
   "Unit1.Em7.ControlNodes".cm.Command.jrWinderAxisB.posAbsolute[4] := #_w1;
END_REGION

REGION Network 208: CmJRWinderAxisB Position Absolute Position5
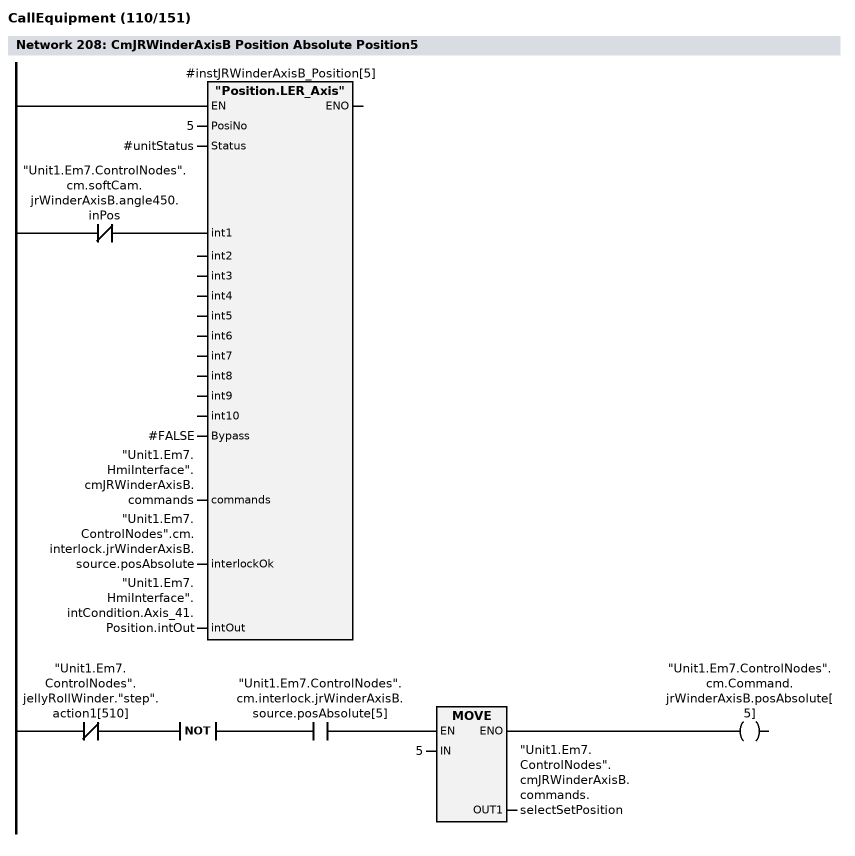
   RUNG wire#powerrail
      #instJRWinderAxisB_Position[5](int1 := wire#w1, PosiNo := 5, Status := #unitStatus, int2 :=, int3 :=, int4 :=, int5 :=, int6 :=, int7 :=, int8 :=, int9 :=, int10 :=, Bypass := #FALSE, commands := "Unit1.Em7.HmiInterface".cmJRWinderAxisB.commands, interlockOk := "Unit1.Em7.ControlNodes".cm.interlock.jrWinderAxisB.source.posAbsolute, intOut := "Unit1.Em7.HmiInterface".intCondition.Axis_41.Position.intOut)
   END_RUNG
   RUNG wire#powerrail
      I_Contact( "Unit1.Em7.ControlNodes".cm.softCam.jrWinderAxisB.angle450.inPos )
   END_RUNG wire#w1
   RUNG wire#powerrail
      I_Contact( "Unit1.Em7.ControlNodes".jellyRollWinder."step".action1[510] )
      Not()
      Contact( "Unit1.Em7.ControlNodes".cm.interlock.jrWinderAxisB.source.posAbsolute[5] )
      Move(in := 5, out1 => "Unit1.Em7.ControlNodes".cmJRWinderAxisB.commands.selectSetPosition)
      Coil( "Unit1.Em7.ControlNodes".cm.Command.jrWinderAxisB.posAbsolute[5] )
   END_RUNG
   // the same network as SCL:
   #instJRWinderAxisB_Position[5](PosiNo := 5,   // "Position.LER_Axis"
                           Status := #unitStatus,
                           int1 := NOT "Unit1.Em7.ControlNodes".cm.softCam.jrWinderAxisB.angle450.inPos,
                           Bypass := #FALSE,
                           commands := "Unit1.Em7.HmiInterface".cmJRWinderAxisB.commands,
                           interlockOk := "Unit1.Em7.ControlNodes".cm.interlock.jrWinderAxisB.source.posAbsolute,
                           intOut := "Unit1.Em7.HmiInterface".intCondition.Axis_41.Position.intOut);
   #_w1 := NOT (NOT "Unit1.Em7.ControlNodes".jellyRollWinder."step".action1[510]) AND "Unit1.Em7.ControlNodes".cm.interlock.jrWinderAxisB.source.posAbsolute[5];
   IF #_w1 THEN "Unit1.Em7.ControlNodes".cmJRWinderAxisB.commands.selectSetPosition := 5; END_IF;
   "Unit1.Em7.ControlNodes".cm.Command.jrWinderAxisB.posAbsolute[5] := #_w1;
END_REGION

REGION Network 209: CmJRWinderAxisB Position Absolute Position6
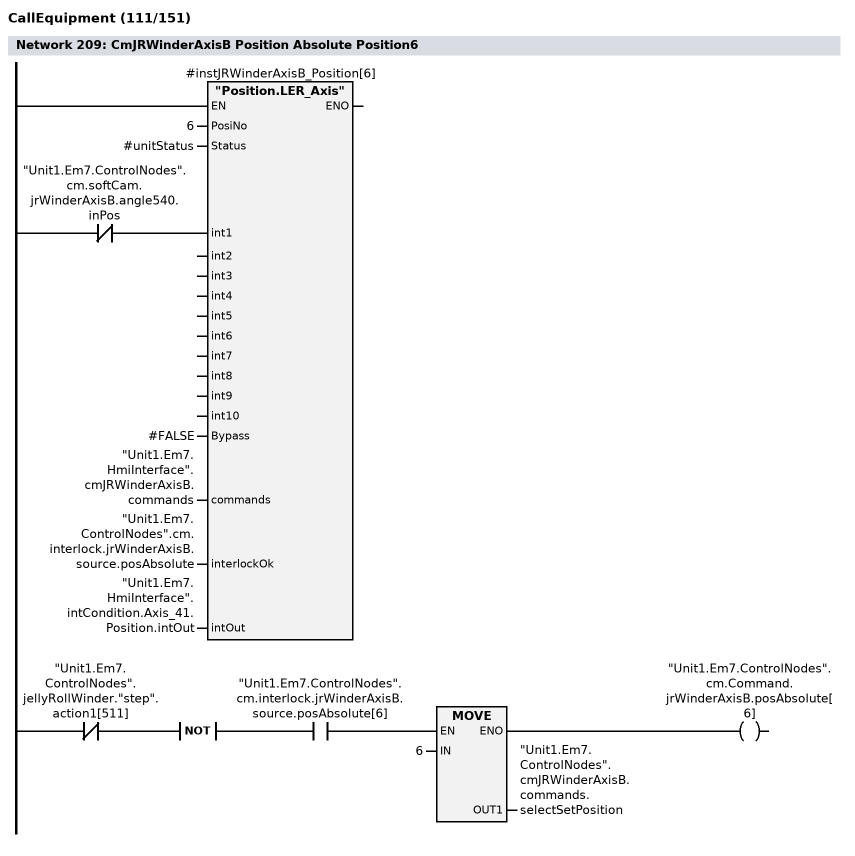
   RUNG wire#powerrail
      #instJRWinderAxisB_Position[6](int1 := wire#w1, PosiNo := 6, Status := #unitStatus, int2 :=, int3 :=, int4 :=, int5 :=, int6 :=, int7 :=, int8 :=, int9 :=, int10 :=, Bypass := #FALSE, commands := "Unit1.Em7.HmiInterface".cmJRWinderAxisB.commands, interlockOk := "Unit1.Em7.ControlNodes".cm.interlock.jrWinderAxisB.source.posAbsolute, intOut := "Unit1.Em7.HmiInterface".intCondition.Axis_41.Position.intOut)
   END_RUNG
   RUNG wire#powerrail
      I_Contact( "Unit1.Em7.ControlNodes".cm.softCam.jrWinderAxisB.angle540.inPos )
   END_RUNG wire#w1
   RUNG wire#powerrail
      I_Contact( "Unit1.Em7.ControlNodes".jellyRollWinder."step".action1[511] )
      Not()
      Contact( "Unit1.Em7.ControlNodes".cm.interlock.jrWinderAxisB.source.posAbsolute[6] )
      Move(in := 6, out1 => "Unit1.Em7.ControlNodes".cmJRWinderAxisB.commands.selectSetPosition)
      Coil( "Unit1.Em7.ControlNodes".cm.Command.jrWinderAxisB.posAbsolute[6] )
   END_RUNG
   // the same network as SCL:
   #instJRWinderAxisB_Position[6](PosiNo := 6,   // "Position.LER_Axis"
                           Status := #unitStatus,
                           int1 := NOT "Unit1.Em7.ControlNodes".cm.softCam.jrWinderAxisB.angle540.inPos,
                           Bypass := #FALSE,
                           commands := "Unit1.Em7.HmiInterface".cmJRWinderAxisB.commands,
                           interlockOk := "Unit1.Em7.ControlNodes".cm.interlock.jrWinderAxisB.source.posAbsolute,
                           intOut := "Unit1.Em7.HmiInterface".intCondition.Axis_41.Position.intOut);
   #_w1 := NOT (NOT "Unit1.Em7.ControlNodes".jellyRollWinder."step".action1[511]) AND "Unit1.Em7.ControlNodes".cm.interlock.jrWinderAxisB.source.posAbsolute[6];
   IF #_w1 THEN "Unit1.Em7.ControlNodes".cmJRWinderAxisB.commands.selectSetPosition := 6; END_IF;
   "Unit1.Em7.ControlNodes".cm.Command.jrWinderAxisB.posAbsolute[6] := #_w1;
END_REGION

REGION Network 210: CmJRWinderAxisB Position Absolute Position7
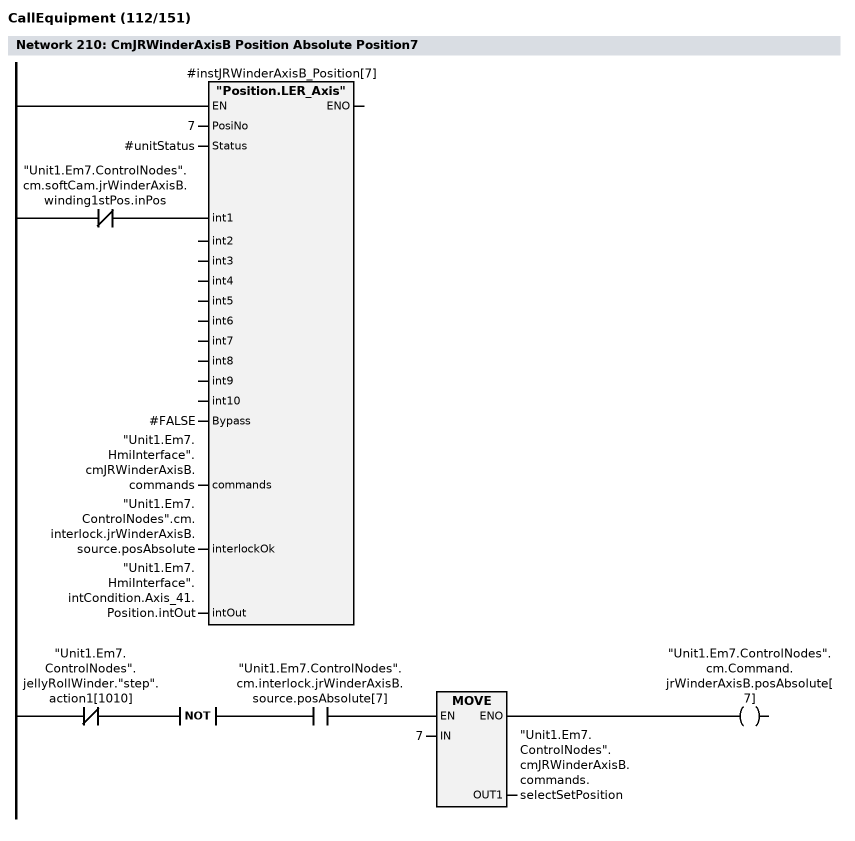
   RUNG wire#powerrail
      #instJRWinderAxisB_Position[7](int1 := wire#w1, PosiNo := 7, Status := #unitStatus, int2 :=, int3 :=, int4 :=, int5 :=, int6 :=, int7 :=, int8 :=, int9 :=, int10 :=, Bypass := #FALSE, commands := "Unit1.Em7.HmiInterface".cmJRWinderAxisB.commands, interlockOk := "Unit1.Em7.ControlNodes".cm.interlock.jrWinderAxisB.source.posAbsolute, intOut := "Unit1.Em7.HmiInterface".intCondition.Axis_41.Position.intOut)
   END_RUNG
   RUNG wire#powerrail
      I_Contact( "Unit1.Em7.ControlNodes".cm.softCam.jrWinderAxisB.winding1stPos.inPos )
   END_RUNG wire#w1
   RUNG wire#powerrail
      I_Contact( "Unit1.Em7.ControlNodes".jellyRollWinder."step".action1[1010] )
      Not()
      Contact( "Unit1.Em7.ControlNodes".cm.interlock.jrWinderAxisB.source.posAbsolute[7] )
      Move(in := 7, out1 => "Unit1.Em7.ControlNodes".cmJRWinderAxisB.commands.selectSetPosition)
      Coil( "Unit1.Em7.ControlNodes".cm.Command.jrWinderAxisB.posAbsolute[7] )
   END_RUNG
   // the same network as SCL:
   #instJRWinderAxisB_Position[7](PosiNo := 7,   // "Position.LER_Axis"
                           Status := #unitStatus,
                           int1 := NOT "Unit1.Em7.ControlNodes".cm.softCam.jrWinderAxisB.winding1stPos.inPos,
                           Bypass := #FALSE,
                           commands := "Unit1.Em7.HmiInterface".cmJRWinderAxisB.commands,
                           interlockOk := "Unit1.Em7.ControlNodes".cm.interlock.jrWinderAxisB.source.posAbsolute,
                           intOut := "Unit1.Em7.HmiInterface".intCondition.Axis_41.Position.intOut);
   #_w1 := NOT (NOT "Unit1.Em7.ControlNodes".jellyRollWinder."step".action1[1010]) AND "Unit1.Em7.ControlNodes".cm.interlock.jrWinderAxisB.source.posAbsolute[7];
   IF #_w1 THEN "Unit1.Em7.ControlNodes".cmJRWinderAxisB.commands.selectSetPosition := 7; END_IF;
   "Unit1.Em7.ControlNodes".cm.Command.jrWinderAxisB.posAbsolute[7] := #_w1;
END_REGION

REGION Network 211: CmJRWinderAxisB Position Absolute Position8
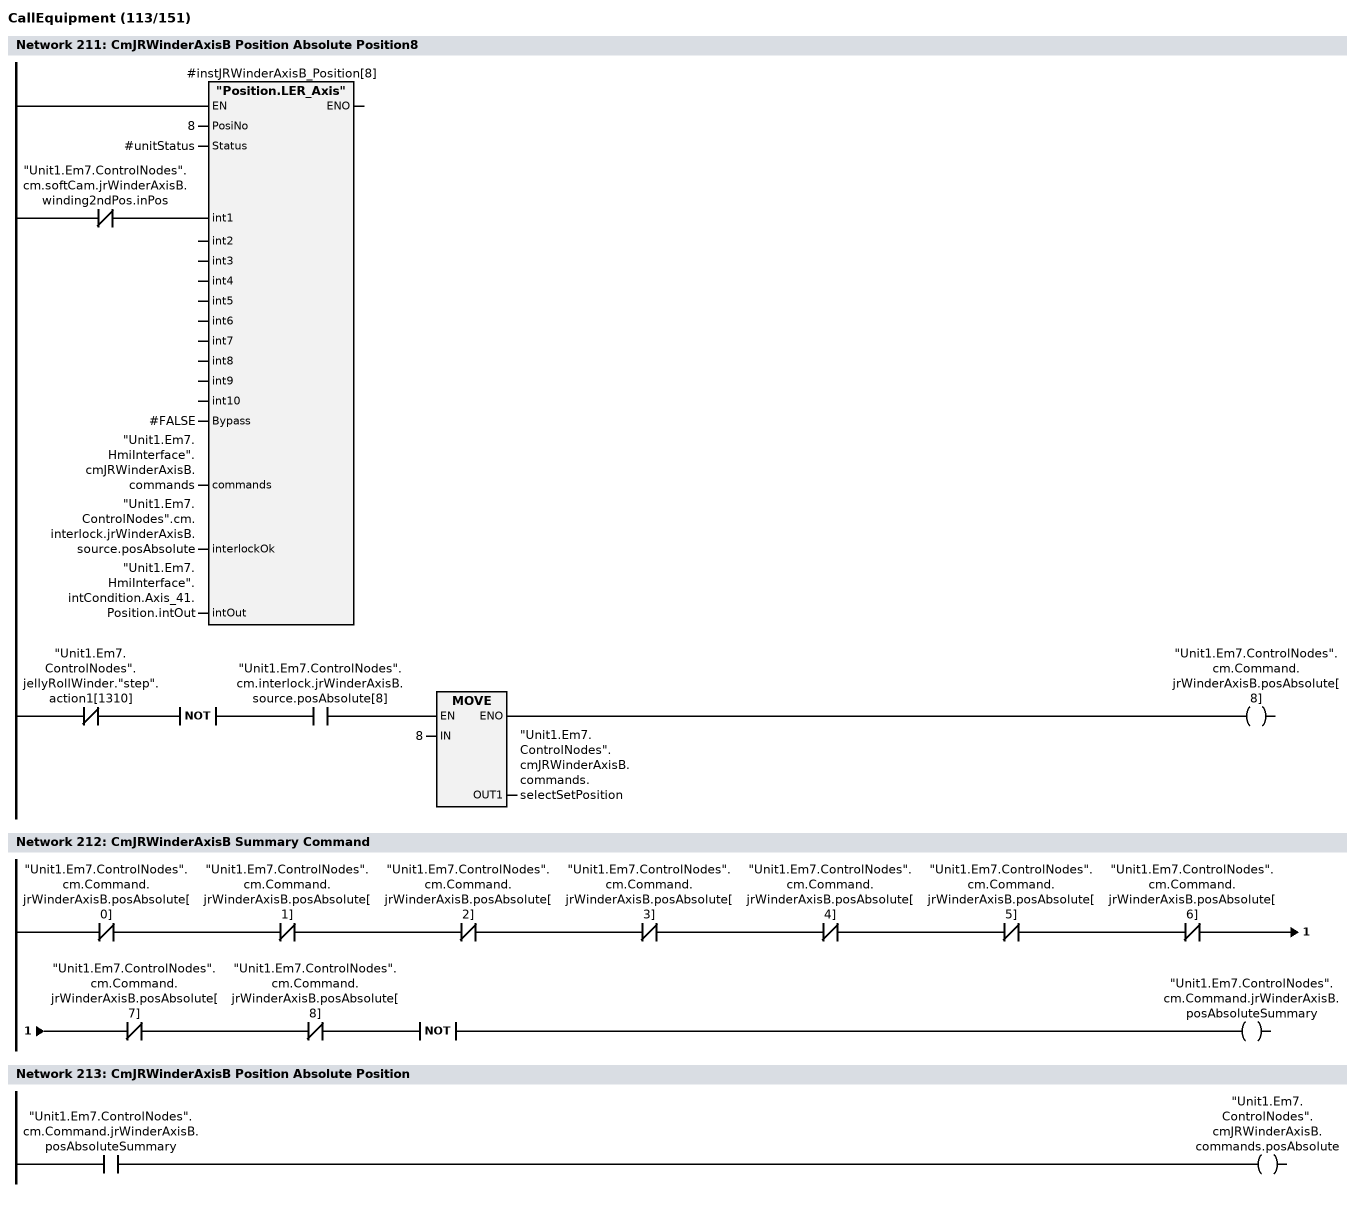
   RUNG wire#powerrail
      #instJRWinderAxisB_Position[8](int1 := wire#w1, PosiNo := 8, Status := #unitStatus, int2 :=, int3 :=, int4 :=, int5 :=, int6 :=, int7 :=, int8 :=, int9 :=, int10 :=, Bypass := #FALSE, commands := "Unit1.Em7.HmiInterface".cmJRWinderAxisB.commands, interlockOk := "Unit1.Em7.ControlNodes".cm.interlock.jrWinderAxisB.source.posAbsolute, intOut := "Unit1.Em7.HmiInterface".intCondition.Axis_41.Position.intOut)
   END_RUNG
   RUNG wire#powerrail
      I_Contact( "Unit1.Em7.ControlNodes".cm.softCam.jrWinderAxisB.winding2ndPos.inPos )
   END_RUNG wire#w1
   RUNG wire#powerrail
      I_Contact( "Unit1.Em7.ControlNodes".jellyRollWinder."step".action1[1310] )
      Not()
      Contact( "Unit1.Em7.ControlNodes".cm.interlock.jrWinderAxisB.source.posAbsolute[8] )
      Move(in := 8, out1 => "Unit1.Em7.ControlNodes".cmJRWinderAxisB.commands.selectSetPosition)
      Coil( "Unit1.Em7.ControlNodes".cm.Command.jrWinderAxisB.posAbsolute[8] )
   END_RUNG
   // the same network as SCL:
   #instJRWinderAxisB_Position[8](PosiNo := 8,   // "Position.LER_Axis"
                           Status := #unitStatus,
                           int1 := NOT "Unit1.Em7.ControlNodes".cm.softCam.jrWinderAxisB.winding2ndPos.inPos,
                           Bypass := #FALSE,
                           commands := "Unit1.Em7.HmiInterface".cmJRWinderAxisB.commands,
                           interlockOk := "Unit1.Em7.ControlNodes".cm.interlock.jrWinderAxisB.source.posAbsolute,
                           intOut := "Unit1.Em7.HmiInterface".intCondition.Axis_41.Position.intOut);
   #_w1 := NOT (NOT "Unit1.Em7.ControlNodes".jellyRollWinder."step".action1[1310]) AND "Unit1.Em7.ControlNodes".cm.interlock.jrWinderAxisB.source.posAbsolute[8];
   IF #_w1 THEN "Unit1.Em7.ControlNodes".cmJRWinderAxisB.commands.selectSetPosition := 8; END_IF;
   "Unit1.Em7.ControlNodes".cm.Command.jrWinderAxisB.posAbsolute[8] := #_w1;
END_REGION

REGION Network 212: CmJRWinderAxisB Summary Command
   RUNG wire#powerrail
      I_Contact( "Unit1.Em7.ControlNodes".cm.Command.jrWinderAxisB.posAbsolute[0] )
      I_Contact( "Unit1.Em7.ControlNodes".cm.Command.jrWinderAxisB.posAbsolute[1] )
      I_Contact( "Unit1.Em7.ControlNodes".cm.Command.jrWinderAxisB.posAbsolute[2] )
      I_Contact( "Unit1.Em7.ControlNodes".cm.Command.jrWinderAxisB.posAbsolute[3] )
      I_Contact( "Unit1.Em7.ControlNodes".cm.Command.jrWinderAxisB.posAbsolute[4] )
      I_Contact( "Unit1.Em7.ControlNodes".cm.Command.jrWinderAxisB.posAbsolute[5] )
      I_Contact( "Unit1.Em7.ControlNodes".cm.Command.jrWinderAxisB.posAbsolute[6] )
      I_Contact( "Unit1.Em7.ControlNodes".cm.Command.jrWinderAxisB.posAbsolute[7] )
      I_Contact( "Unit1.Em7.ControlNodes".cm.Command.jrWinderAxisB.posAbsolute[8] )
      Not()
      Coil( "Unit1.Em7.ControlNodes".cm.Command.jrWinderAxisB.posAbsoluteSummary )
   END_RUNG
   // the same network as SCL:
   "Unit1.Em7.ControlNodes".cm.Command.jrWinderAxisB.posAbsoluteSummary := NOT (NOT "Unit1.Em7.ControlNodes".cm.Command.jrWinderAxisB.posAbsolute[0] AND NOT "Unit1.Em7.ControlNodes".cm.Command.jrWinderAxisB.posAbsolute[1] AND NOT "Unit1.Em7.ControlNodes".cm.Command.jrWinderAxisB.posAbsolute[2] AND NOT "Unit1.Em7.ControlNodes".cm.Command.jrWinderAxisB.posAbsolute[3] AND NOT "Unit1.Em7.ControlNodes".cm.Command.jrWinderAxisB.posAbsolute[4] AND NOT "Unit1.Em7.ControlNodes".cm.Command.jrWinderAxisB.posAbsolute[5] AND NOT "Unit1.Em7.ControlNodes".cm.Command.jrWinderAxisB.posAbsolute[6] AND NOT "Unit1.Em7.ControlNodes".cm.Command.jrWinderAxisB.posAbsolute[7] AND NOT "Unit1.Em7.ControlNodes".cm.Command.jrWinderAxisB.posAbsolute[8]);
END_REGION

REGION Network 213: CmJRWinderAxisB Position Absolute Position
   RUNG wire#powerrail
      Contact( "Unit1.Em7.ControlNodes".cm.Command.jrWinderAxisB.posAbsoluteSummary )
      Coil( "Unit1.Em7.ControlNodes".cmJRWinderAxisB.commands.posAbsolute )
   END_RUNG
   // the same network as SCL:
   "Unit1.Em7.ControlNodes".cmJRWinderAxisB.commands.posAbsolute := "Unit1.Em7.ControlNodes".cm.Command.jrWinderAxisB.posAbsoluteSummary;
END_REGION

REGION Network 214: CmJRWinderAxisB Interlock Summary
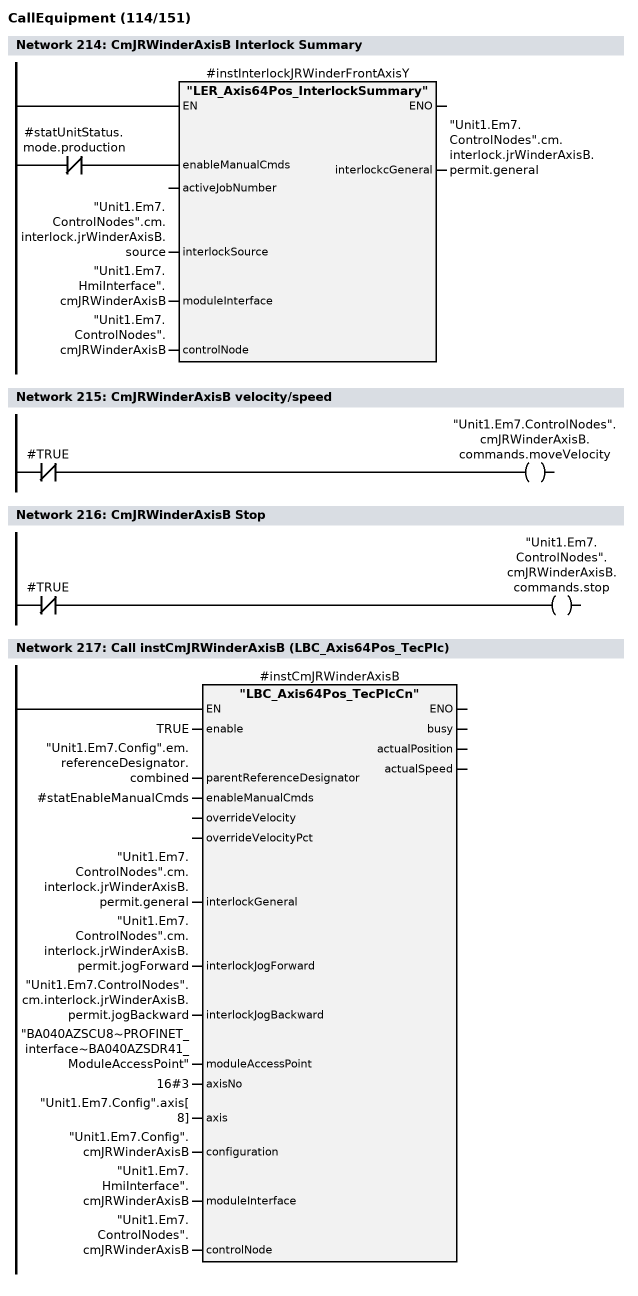
   RUNG wire#powerrail
      #instInterlockJRWinderFrontAxisY(enableManualCmds := wire#w1, activeJobNumber :=, interlockSource := "Unit1.Em7.ControlNodes".cm.interlock.jrWinderAxisB.source, moduleInterface := "Unit1.Em7.HmiInterface".cmJRWinderAxisB, controlNode := "Unit1.Em7.ControlNodes".cmJRWinderAxisB, interlockcGeneral => "Unit1.Em7.ControlNodes".cm.interlock.jrWinderAxisB.permit.general)
   END_RUNG
   RUNG wire#powerrail
      I_Contact( #statUnitStatus.mode.production )
   END_RUNG wire#w1
   // the same network as SCL:
   #instInterlockJRWinderFrontAxisY(enableManualCmds := NOT #statUnitStatus.mode.production,   // "LER_Axis64Pos_InterlockSummary"
                           interlockSource := "Unit1.Em7.ControlNodes".cm.interlock.jrWinderAxisB.source,
                           moduleInterface := "Unit1.Em7.HmiInterface".cmJRWinderAxisB,
                           controlNode := "Unit1.Em7.ControlNodes".cmJRWinderAxisB,
                           interlockcGeneral => "Unit1.Em7.ControlNodes".cm.interlock.jrWinderAxisB.permit.general);
END_REGION

REGION Network 215: CmJRWinderAxisB velocity/speed
   RUNG wire#powerrail
      I_Contact( #TRUE )
      Coil( "Unit1.Em7.ControlNodes".cmJRWinderAxisB.commands.moveVelocity )
   END_RUNG
   // the same network as SCL:
   "Unit1.Em7.ControlNodes".cmJRWinderAxisB.commands.moveVelocity := NOT #TRUE;
END_REGION

REGION Network 216: CmJRWinderAxisB Stop
   RUNG wire#powerrail
      I_Contact( #TRUE )
      Coil( "Unit1.Em7.ControlNodes".cmJRWinderAxisB.commands.stop )
   END_RUNG
   // the same network as SCL:
   "Unit1.Em7.ControlNodes".cmJRWinderAxisB.commands.stop := NOT #TRUE;
END_REGION

REGION Network 217: Call instCmJRWinderAxisB (LBC_Axis64Pos_TecPlc)
   RUNG wire#powerrail
      #instCmJRWinderAxisB(enable := TRUE, parentReferenceDesignator := "Unit1.Em7.Config".em.referenceDesignator.combined, enableManualCmds := #statEnableManualCmds, overrideVelocity :=, overrideVelocityPct :=, interlockGeneral := "Unit1.Em7.ControlNodes".cm.interlock.jrWinderAxisB.permit.general, interlockJogForward := "Unit1.Em7.ControlNodes".cm.interlock.jrWinderAxisB.permit.jogForward, interlockJogBackward := "Unit1.Em7.ControlNodes".cm.interlock.jrWinderAxisB.permit.jogBackward, moduleAccessPoint := "BA040AZSCU8~PROFINET_interface~BA040AZSDR41_ModuleAccessPoint", axisNo := 16#3, axis := "Unit1.Em7.Config".axis[8], configuration := "Unit1.Em7.Config".cmJRWinderAxisB, moduleInterface := "Unit1.Em7.HmiInterface".cmJRWinderAxisB, controlNode := "Unit1.Em7.ControlNodes".cmJRWinderAxisB, busy =>, actualPosition =>, actualSpeed =>)
   END_RUNG
   // the same network as SCL:
   #instCmJRWinderAxisB(enable := TRUE,   // "LBC_Axis64Pos_TecPlcCn"
                        parentReferenceDesignator := "Unit1.Em7.Config".em.referenceDesignator.combined,
                        enableManualCmds := #statEnableManualCmds,
                        interlockGeneral := "Unit1.Em7.ControlNodes".cm.interlock.jrWinderAxisB.permit.general,
                        interlockJogForward := "Unit1.Em7.ControlNodes".cm.interlock.jrWinderAxisB.permit.jogForward,
                        interlockJogBackward := "Unit1.Em7.ControlNodes".cm.interlock.jrWinderAxisB.permit.jogBackward,
                        moduleAccessPoint := "BA040AZSCU8~PROFINET_interface~BA040AZSDR41_ModuleAccessPoint",
                        axisNo := 16#3,
                        axis := "Unit1.Em7.Config".axis[8],
                        configuration := "Unit1.Em7.Config".cmJRWinderAxisB,
                        moduleInterface := "Unit1.Em7.HmiInterface".cmJRWinderAxisB,
                        controlNode := "Unit1.Em7.ControlNodes".cmJRWinderAxisB);
END_REGION

REGION Network 218: JRWinderAxisB SoftCam
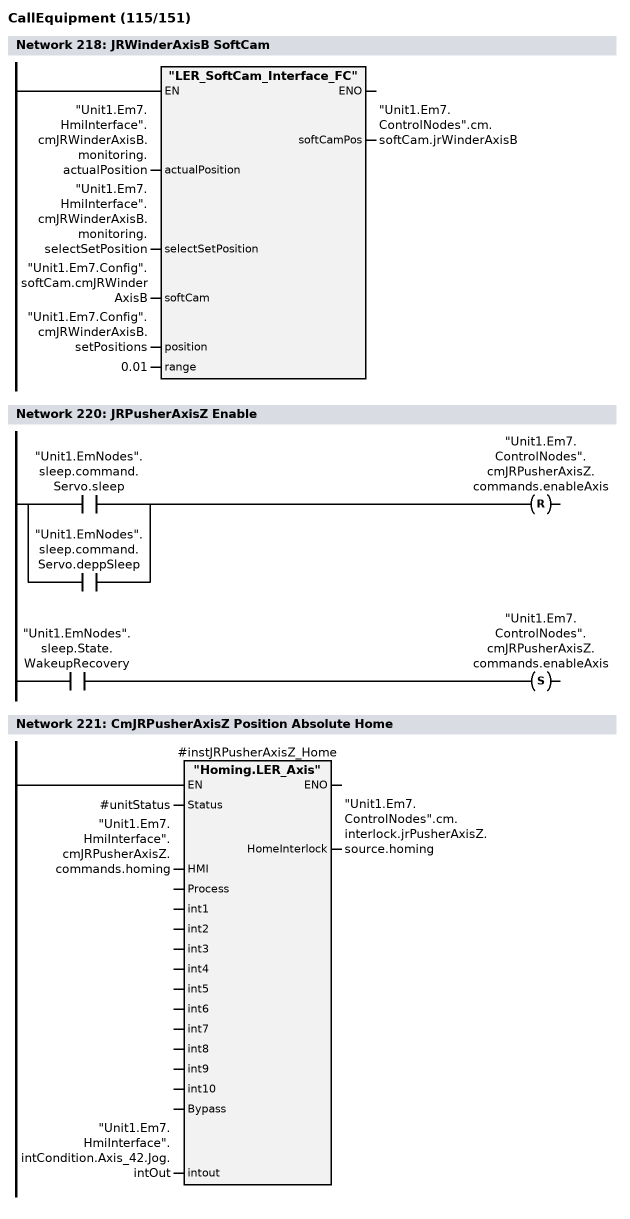
   RUNG wire#powerrail
      "LER_SoftCam_Interface_FC"(actualPosition := "Unit1.Em7.HmiInterface".cmJRWinderAxisB.monitoring.actualPosition, selectSetPosition := "Unit1.Em7.HmiInterface".cmJRWinderAxisB.monitoring.selectSetPosition, softCam := "Unit1.Em7.Config".softCam.cmJRWinderAxisB, position := "Unit1.Em7.Config".cmJRWinderAxisB.setPositions, range := 0.01, softCamPos => "Unit1.Em7.ControlNodes".cm.softCam.jrWinderAxisB)
   END_RUNG
   // the same network as SCL:
   "LER_SoftCam_Interface_FC"(actualPosition := "Unit1.Em7.HmiInterface".cmJRWinderAxisB.monitoring.actualPosition,
                           selectSetPosition := "Unit1.Em7.HmiInterface".cmJRWinderAxisB.monitoring.selectSetPosition,
                           softCam := "Unit1.Em7.Config".softCam.cmJRWinderAxisB,
                           position := "Unit1.Em7.Config".cmJRWinderAxisB.setPositions,
                           range := 0.01,
                           softCamPos => "Unit1.Em7.ControlNodes".cm.softCam.jrWinderAxisB);
END_REGION

REGION Network 220: JRPusherAxisZ Enable
   RUNG wire#powerrail
      Contact( "Unit1.EmNodes".sleep.command.Servo.sleep )
      wire#w1
      R_Coil( "Unit1.Em7.ControlNodes".cmJRPusherAxisZ.commands.enableAxis )
   END_RUNG
   RUNG wire#powerrail
      Contact( "Unit1.EmNodes".sleep.command.Servo.deppSleep )
   END_RUNG wire#w1
   RUNG wire#powerrail
      Contact( "Unit1.EmNodes".sleep.State.WakeupRecovery )
      S_Coil( "Unit1.Em7.ControlNodes".cmJRPusherAxisZ.commands.enableAxis )
   END_RUNG
   // the same network as SCL:
   IF "Unit1.EmNodes".sleep.command.Servo.sleep OR "Unit1.EmNodes".sleep.command.Servo.deppSleep THEN
       "Unit1.Em7.ControlNodes".cmJRPusherAxisZ.commands.enableAxis := FALSE;
   END_IF;
   IF "Unit1.EmNodes".sleep.State.WakeupRecovery THEN
       "Unit1.Em7.ControlNodes".cmJRPusherAxisZ.commands.enableAxis := TRUE;
   END_IF;
END_REGION

REGION Network 221: CmJRPusherAxisZ Position Absolute Home
   RUNG wire#powerrail
      #instJRPusherAxisZ_Home(Status := #unitStatus, HMI := "Unit1.Em7.HmiInterface".cmJRPusherAxisZ.commands.homing, Process :=, int1 :=, int2 :=, int3 :=, int4 :=, int5 :=, int6 :=, int7 :=, int8 :=, int9 :=, int10 :=, Bypass :=, intout := "Unit1.Em7.HmiInterface".intCondition.Axis_42.Jog.intOut, HomeInterlock => "Unit1.Em7.ControlNodes".cm.interlock.jrPusherAxisZ.source.homing)
   END_RUNG
   // the same network as SCL:
   #instJRPusherAxisZ_Home(Status := #unitStatus,   // "Homing.LER_Axis"
                           HMI := "Unit1.Em7.HmiInterface".cmJRPusherAxisZ.commands.homing,
                           intout := "Unit1.Em7.HmiInterface".intCondition.Axis_42.Jog.intOut,
                           HomeInterlock => "Unit1.Em7.ControlNodes".cm.interlock.jrPusherAxisZ.source.homing);
END_REGION

REGION Network 222: CmJRPusherAxisZ Position Absolute Jog
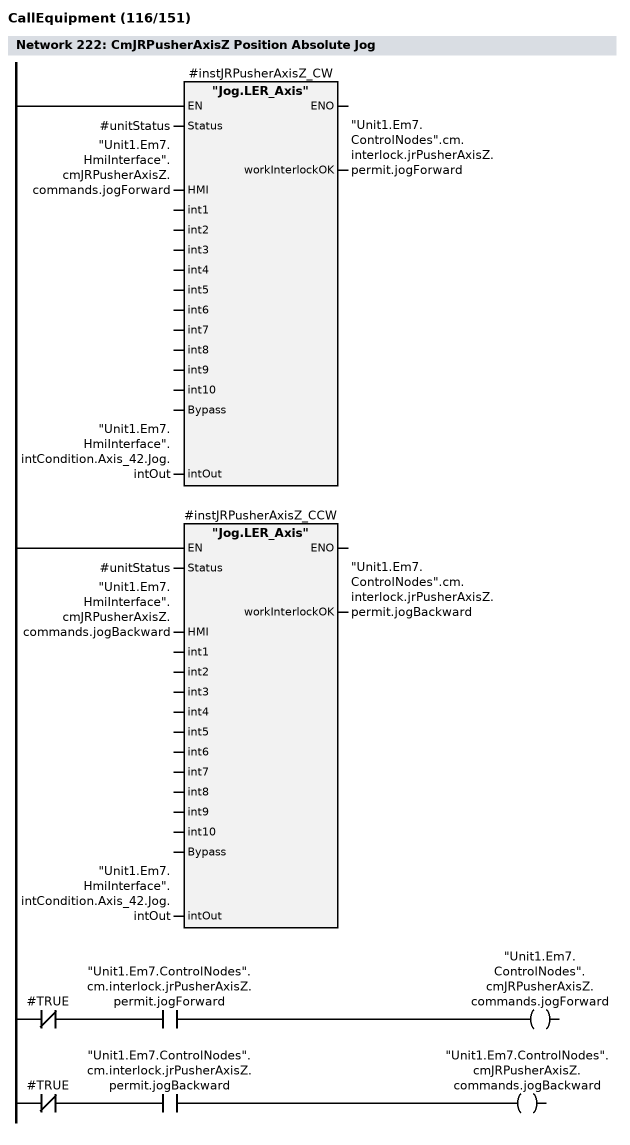
   RUNG wire#powerrail
      #instJRPusherAxisZ_CW(Status := #unitStatus, HMI := "Unit1.Em7.HmiInterface".cmJRPusherAxisZ.commands.jogForward, int1 :=, int2 :=, int3 :=, int4 :=, int5 :=, int6 :=, int7 :=, int8 :=, int9 :=, int10 :=, Bypass :=, intOut := "Unit1.Em7.HmiInterface".intCondition.Axis_42.Jog.intOut, workInterlockOK => "Unit1.Em7.ControlNodes".cm.interlock.jrPusherAxisZ.permit.jogForward)
   END_RUNG
   RUNG wire#powerrail
      #instJRPusherAxisZ_CCW(Status := #unitStatus, HMI := "Unit1.Em7.HmiInterface".cmJRPusherAxisZ.commands.jogBackward, int1 :=, int2 :=, int3 :=, int4 :=, int5 :=, int6 :=, int7 :=, int8 :=, int9 :=, int10 :=, Bypass :=, intOut := "Unit1.Em7.HmiInterface".intCondition.Axis_42.Jog.intOut, workInterlockOK => "Unit1.Em7.ControlNodes".cm.interlock.jrPusherAxisZ.permit.jogBackward)
   END_RUNG
   RUNG wire#powerrail
      I_Contact( #TRUE )
      Contact( "Unit1.Em7.ControlNodes".cm.interlock.jrPusherAxisZ.permit.jogForward )
      Coil( "Unit1.Em7.ControlNodes".cmJRPusherAxisZ.commands.jogForward )
   END_RUNG
   RUNG wire#powerrail
      I_Contact( #TRUE )
      Contact( "Unit1.Em7.ControlNodes".cm.interlock.jrPusherAxisZ.permit.jogBackward )
      Coil( "Unit1.Em7.ControlNodes".cmJRPusherAxisZ.commands.jogBackward )
   END_RUNG
   // the same network as SCL:
   #instJRPusherAxisZ_CW(Status := #unitStatus,   // "Jog.LER_Axis"
                         HMI := "Unit1.Em7.HmiInterface".cmJRPusherAxisZ.commands.jogForward,
                         intOut := "Unit1.Em7.HmiInterface".intCondition.Axis_42.Jog.intOut,
                         workInterlockOK => "Unit1.Em7.ControlNodes".cm.interlock.jrPusherAxisZ.permit.jogForward);
   #instJRPusherAxisZ_CCW(Status := #unitStatus,   // "Jog.LER_Axis"
                          HMI := "Unit1.Em7.HmiInterface".cmJRPusherAxisZ.commands.jogBackward,
                          intOut := "Unit1.Em7.HmiInterface".intCondition.Axis_42.Jog.intOut,
                          workInterlockOK => "Unit1.Em7.ControlNodes".cm.interlock.jrPusherAxisZ.permit.jogBackward);
   "Unit1.Em7.ControlNodes".cmJRPusherAxisZ.commands.jogForward := NOT #TRUE AND "Unit1.Em7.ControlNodes".cm.interlock.jrPusherAxisZ.permit.jogForward;
   "Unit1.Em7.ControlNodes".cmJRPusherAxisZ.commands.jogBackward := NOT #TRUE AND "Unit1.Em7.ControlNodes".cm.interlock.jrPusherAxisZ.permit.jogBackward;
END_REGION

REGION Network 223: CmJRPusherAxisZ Position Absolute Position0
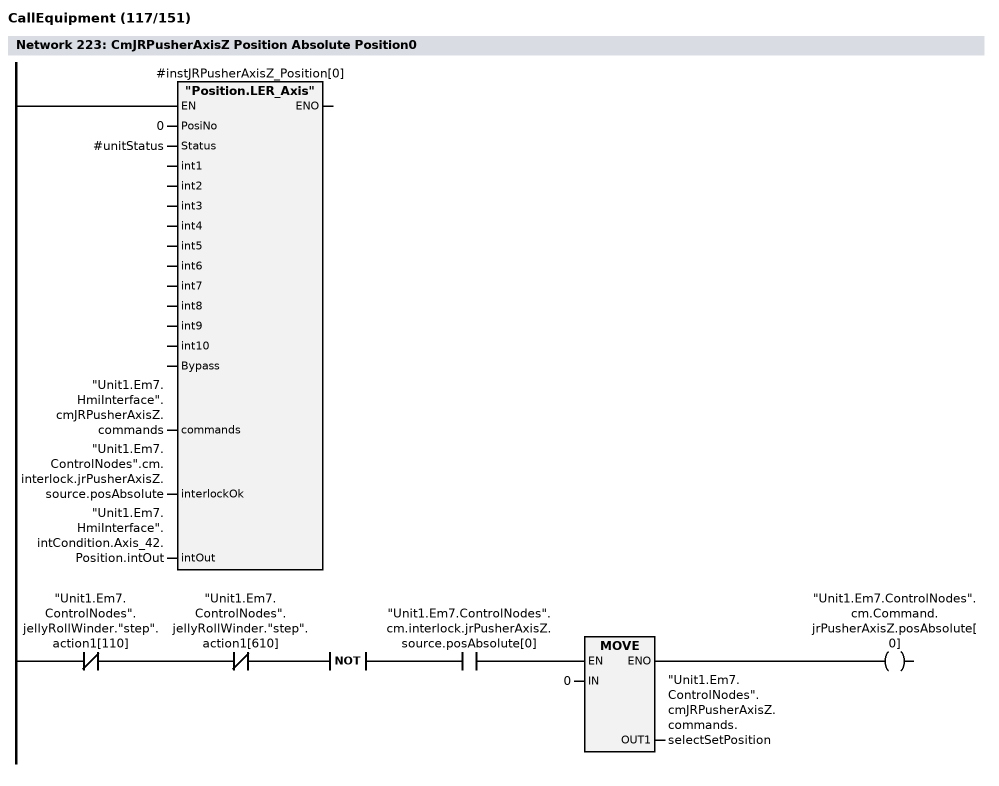
   RUNG wire#powerrail
      #instJRPusherAxisZ_Position[0](PosiNo := 0, Status := #unitStatus, int1 :=, int2 :=, int3 :=, int4 :=, int5 :=, int6 :=, int7 :=, int8 :=, int9 :=, int10 :=, Bypass :=, commands := "Unit1.Em7.HmiInterface".cmJRPusherAxisZ.commands, interlockOk := "Unit1.Em7.ControlNodes".cm.interlock.jrPusherAxisZ.source.posAbsolute, intOut := "Unit1.Em7.HmiInterface".intCondition.Axis_42.Position.intOut)
   END_RUNG
   RUNG wire#powerrail
      I_Contact( "Unit1.Em7.ControlNodes".jellyRollWinder."step".action1[110] )
      I_Contact( "Unit1.Em7.ControlNodes".jellyRollWinder."step".action1[610] )
      Not()
      Contact( "Unit1.Em7.ControlNodes".cm.interlock.jrPusherAxisZ.source.posAbsolute[0] )
      Move(in := 0, out1 => "Unit1.Em7.ControlNodes".cmJRPusherAxisZ.commands.selectSetPosition)
      Coil( "Unit1.Em7.ControlNodes".cm.Command.jrPusherAxisZ.posAbsolute[0] )
   END_RUNG
   // the same network as SCL:
   #instJRPusherAxisZ_Position[0](PosiNo := 0,   // "Position.LER_Axis"
                           Status := #unitStatus,
                           commands := "Unit1.Em7.HmiInterface".cmJRPusherAxisZ.commands,
                           interlockOk := "Unit1.Em7.ControlNodes".cm.interlock.jrPusherAxisZ.source.posAbsolute,
                           intOut := "Unit1.Em7.HmiInterface".intCondition.Axis_42.Position.intOut);
   #_w1 := NOT (NOT "Unit1.Em7.ControlNodes".jellyRollWinder."step".action1[110] AND NOT "Unit1.Em7.ControlNodes".jellyRollWinder."step".action1[610]) AND "Unit1.Em7.ControlNodes".cm.interlock.jrPusherAxisZ.source.posAbsolute[0];
   IF #_w1 THEN "Unit1.Em7.ControlNodes".cmJRPusherAxisZ.commands.selectSetPosition := 0; END_IF;
   "Unit1.Em7.ControlNodes".cm.Command.jrPusherAxisZ.posAbsolute[0] := #_w1;
END_REGION

REGION Network 224: CmJRPusherAxisZ Position Absolute Position1
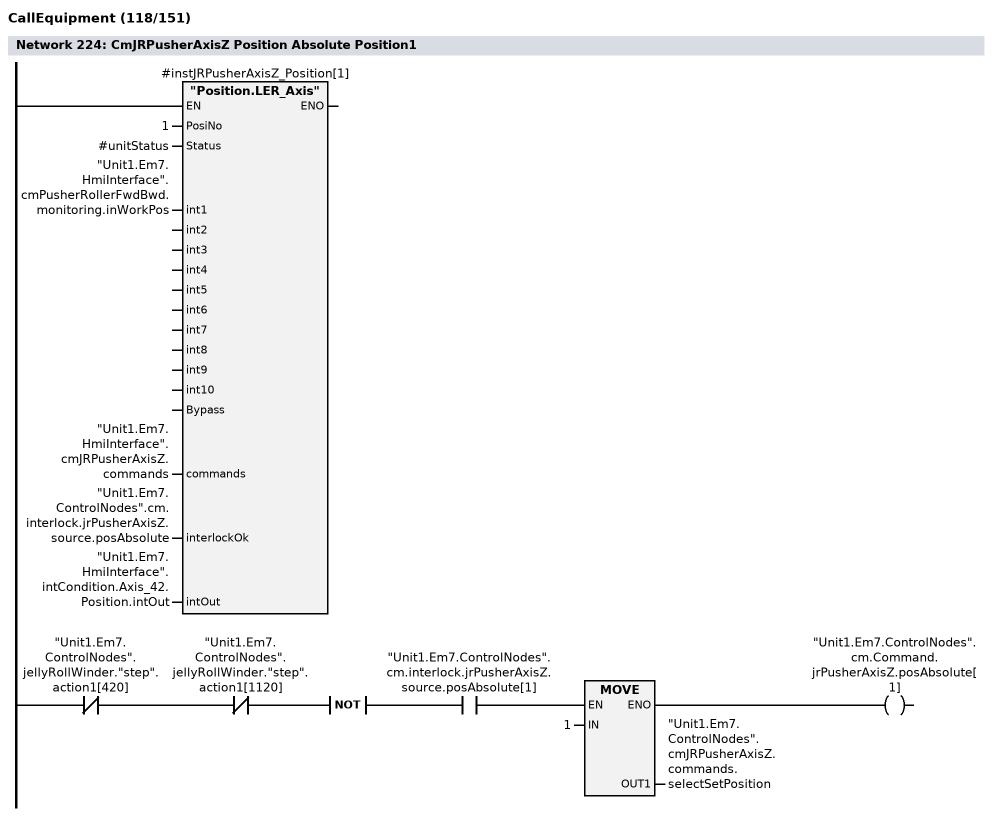
   RUNG wire#powerrail
      #instJRPusherAxisZ_Position[1](PosiNo := 1, Status := #unitStatus, int1 := "Unit1.Em7.HmiInterface".cmPusherRollerFwdBwd.monitoring.inWorkPos, int2 :=, int3 :=, int4 :=, int5 :=, int6 :=, int7 :=, int8 :=, int9 :=, int10 :=, Bypass :=, commands := "Unit1.Em7.HmiInterface".cmJRPusherAxisZ.commands, interlockOk := "Unit1.Em7.ControlNodes".cm.interlock.jrPusherAxisZ.source.posAbsolute, intOut := "Unit1.Em7.HmiInterface".intCondition.Axis_42.Position.intOut)
   END_RUNG
   RUNG wire#powerrail
      I_Contact( "Unit1.Em7.ControlNodes".jellyRollWinder."step".action1[420] )
      I_Contact( "Unit1.Em7.ControlNodes".jellyRollWinder."step".action1[1120] )
      Not()
      Contact( "Unit1.Em7.ControlNodes".cm.interlock.jrPusherAxisZ.source.posAbsolute[1] )
      Move(in := 1, out1 => "Unit1.Em7.ControlNodes".cmJRPusherAxisZ.commands.selectSetPosition)
      Coil( "Unit1.Em7.ControlNodes".cm.Command.jrPusherAxisZ.posAbsolute[1] )
   END_RUNG
   // the same network as SCL:
   #instJRPusherAxisZ_Position[1](PosiNo := 1,   // "Position.LER_Axis"
                           Status := #unitStatus,
                           int1 := "Unit1.Em7.HmiInterface".cmPusherRollerFwdBwd.monitoring.inWorkPos,
                           commands := "Unit1.Em7.HmiInterface".cmJRPusherAxisZ.commands,
                           interlockOk := "Unit1.Em7.ControlNodes".cm.interlock.jrPusherAxisZ.source.posAbsolute,
                           intOut := "Unit1.Em7.HmiInterface".intCondition.Axis_42.Position.intOut);
   #_w1 := NOT (NOT "Unit1.Em7.ControlNodes".jellyRollWinder."step".action1[420] AND NOT "Unit1.Em7.ControlNodes".jellyRollWinder."step".action1[1120]) AND "Unit1.Em7.ControlNodes".cm.interlock.jrPusherAxisZ.source.posAbsolute[1];
   IF #_w1 THEN "Unit1.Em7.ControlNodes".cmJRPusherAxisZ.commands.selectSetPosition := 1; END_IF;
   "Unit1.Em7.ControlNodes".cm.Command.jrPusherAxisZ.posAbsolute[1] := #_w1;
END_REGION

REGION Network 225: CmJRPusherAxisZ Position Absolute Position2
